KUKA KRL program: EPS_2_25694_WD02A_A_20260120031658.src

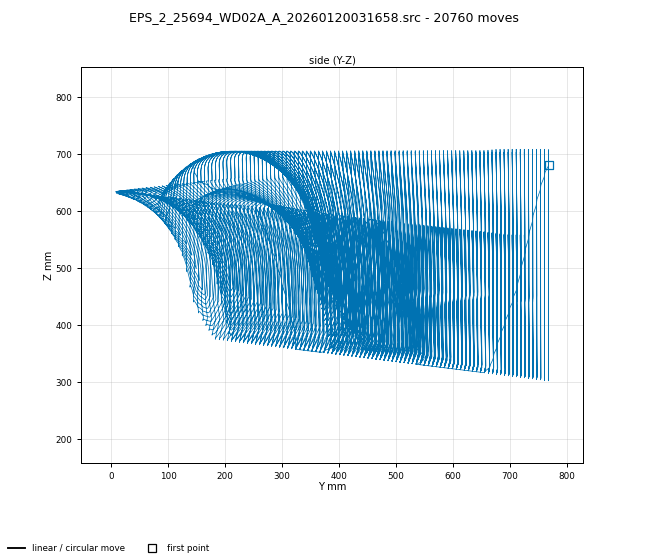
[picture p0: tool path of EPS_2_25694_WD02A_A_20260120031658.src, 20760 of 20762 moves have a stored position in this frame; points joined in program order, loops and branches not executed]
&ACCESS RVP
&REL 4
&COMMENT QRS 19112012
&PARAM EDITMASK = *
DEF PART()
EXT BAS (BAS_COMMAND :IN,REAL :IN )
INT I
BAS (#INITMOV,0 )

;KUKA QRS Post kuka4.cps  Date:22-06-2017 !

File_ID=2999

QRS_PRE_INIT()

;Init var - Until changes are made in qrs_pre_init
Outlet_Square_prg=0
Inlet_1_Square_prg=0
Inlet_2_Square_prg=0
Inlet_3_Square_prg=0
Inlet_4_Square_prg=0
Inlet_5_Square_prg=0

Outlet_1={X 0.000, Y 677.830, Z 583.000, B 0.000, E1 0.000 }
Inlet_1={X 0.000, Y 678.190, Z 578.000, B 0.000, E1 90.000 }
Inlet_2={X 0.000, Y 702.050, Z 243.000, B 0.000, E1 185.000 }
Inlet_3={X 0.000, Y 689.940, Z 413.000, B 0.000, E1 269.000 }
Outlet_1_type=251
Inlet_1_type=251
Inlet_2_type=251
Inlet_3_type=251
;QRS#1=Sidecore dimensions
;QRS#2=250-10" PVC SDR 35
;QRS#3=250-10" PVC SDR 35
;QRS#4=250-10" PVC SDR 35
;QRS#5=250-10" PVC SDR 35
;QRS#6=
;QRS#7=
;QRS#8=
;QRS#9=14M PSX
;QRS#10=14M PSX
;QRS#11=14M PSX
;QRS#12=14M PSX
;QRS#13=
;QRS#14=
;QRS#15=
;QRS#16=1524x152x1067 3,5'
;QRS#17=EPS Height
;QRS#18=708,5
;QRS#19=*
;QRS#20= UPDATED VERSION 22-06-2017
;QRS#21=*
Outlet_Square=0100
Inlet_1_Square=0100
Inlet_2_Square=0100
Inlet_3_Square=0100
Inlet_4_Square=0
Inlet_5_Square=0
Mill_Square=1
Outlet_Square_Prg=205
Inlet_1_Square_prg=205
Inlet_2_Square_prg=205
Inlet_3_Square_prg=205

QRS_INIT()

$ADVANCE=5

; T1
PTP {E1 174.14,E2 174.14}
PTP {X 0,Y 767.497,A -85,B 0,C 180,E1 174.14,E2 174.14,E3 0,E4 0,E5 0,E6 0}
QRS_SPEED_INIT()
LIN {X 0,Y 767.497,Z 681.413,A -85,B 0,C 180,E1 174.14,E2 174.14,E3 0,E4 0,E5 0,E6 0} C_VEL
LIN {X 0,Y 767.498,Z 672.873,A -85,B 0,C 180,E1 173.186,E2 173.186} C_VEL
LIN {X 0,Y 767.497,Z 664.244,A -85,B 0,C 180,E1 172.395,E2 172.395} C_VEL
LIN {X 0,Y 767.496,Z 653.783,A -85,B 0,C 180,E1 171.603,E2 171.603} C_VEL
LIN {X 0,Y 767.499,Z 642.079,A -85,B 0,C 180,E1 170.876,E2 170.876} C_VEL
LIN {X 0,Y 767.47,Z 630.607,A -85,B 0,C 180,E1 170.293,E2 170.293} C_VEL
LIN {X 0,Y 767.488,Z 617.302,A -85,B 0,C 180,E1 169.749,E2 169.749} C_VEL
LIN {X 0,Y 767.494,Z 603.561,A -85,B 0,C 180,E1 169.317,E2 169.317} C_VEL
LIN {X 0,Y 767.478,Z 589.003,A -85,B 0,C 180,E1 168.984,E2 168.984} C_VEL
LIN {X 0,Y 767.456,Z 574.427,A -85,B 0,C 180,E1 168.767,E2 168.767} C_VEL
LIN {X 0,Y 767.491,Z 439.361,A -85,B 0,C 180,E1 167.481,E2 167.481} C_VEL
LIN {X 0,Y 767.485,Z 408.929,A -85,B 0,C 180,E1 164.924,E2 164.924} C_VEL
LIN {X 0,Y 767.474,Z 380.059,A -85,B 0,C 180,E1 162.471,E2 162.471} C_VEL
LIN {X 0,Y 767.471,Z 352.015,A -85,B 0,C 180,E1 160.06,E2 160.06} C_VEL
LIN {X 0,Y 767.448,Z 322.254,A -85,B 0,C 180,E1 157.46,E2 157.46} C_VEL
LIN {X 0,Y 767.468,Z 302.31,A -85,B 0,C 180,E1 155.679,E2 155.679} C_VEL
LIN {X 0,Y 767.445,Z 302.313,A -85,B 0,C 180,E1 153.434,E2 153.434} C_VEL
LIN {X 0,Y 767.444,Z 302.316,A -85,B 0,C 180,E1 151.186,E2 151.186} C_VEL
LIN {X 0,Y 767.451,Z 302.319,A -85,B 0,C 180,E1 149.085,E2 149.085} C_VEL
LIN {X 0,Y 767.479,Z 302.325,A -85,B 0,C 180,E1 146.798,E2 146.798} C_VEL
LIN {X 0,Y 767.488,Z 302.309,A -85,B 0,C 180,E1 144.261,E2 144.261} C_VEL
LIN {X 0,Y 767.459,Z 302.311,A -85,B 0,C 180,E1 141.712,E2 141.712} C_VEL
LIN {X 0,Y 767.472,Z 302.32,A -85,B 0,C 180,E1 139.245,E2 139.245} C_VEL
LIN {X 0,Y 767.481,Z 302.319,A -85,B 0,C 180,E1 136.804,E2 136.804} C_VEL
LIN {X 0,Y 767.479,Z 302.311,A -85,B 0,C 180,E1 134.612,E2 134.612} C_VEL
LIN {X 0,Y 767.493,Z 302.302,A -85,B 0,C 180,E1 132.333,E2 132.333} C_VEL
LIN {X 0,Y 767.47,Z 302.31,A -85,B 0,C 180,E1 129.946,E2 129.946} C_VEL
LIN {X 0,Y 767.489,Z 302.325,A -85,B 0,C 180,E1 127.439,E2 127.439} C_VEL
LIN {X 0,Y 767.472,Z 302.317,A -85,B 0,C 180,E1 125.098,E2 125.098} C_VEL
LIN {X 0,Y 767.487,Z 302.303,A -85,B 0,C 180,E1 122.579,E2 122.579} C_VEL
LIN {X 0,Y 767.485,Z 302.319,A -85,B 0,C 180,E1 119.886,E2 119.886} C_VEL
LIN {X 0,Y 767.49,Z 302.326,A -85,B 0,C 180,E1 117.715,E2 117.715} C_VEL
LIN {X 0,Y 767.461,Z 302.317,A -85,B 0,C 180,E1 115.37,E2 115.37} C_VEL
LIN {X 0,Y 767.457,Z 302.311,A -85,B 0,C 180,E1 113.107,E2 113.107} C_VEL
LIN {X 0,Y 767.471,Z 302.307,A -85,B 0,C 180,E1 110.851,E2 110.851} C_VEL
LIN {X 0,Y 767.488,Z 302.316,A -85,B 0,C 180,E1 108.349,E2 108.349} C_VEL
LIN {X 0,Y 767.466,Z 302.321,A -85,B 0,C 180,E1 105.891,E2 105.891} C_VEL
LIN {X 0,Y 767.447,Z 302.319,A -85,B 0,C 180,E1 103.727,E2 103.727} C_VEL
LIN {X 0,Y 767.436,Z 302.317,A -85,B 0,C 180,E1 101.583,E2 101.583} C_VEL
LIN {X 0,Y 767.437,Z 302.315,A -85,B 0,C 180,E1 99.456,E2 99.456} C_VEL
LIN {X 0,Y 767.443,Z 302.314,A -85,B 0,C 180,E1 97.341,E2 97.341} C_VEL
LIN {X 0,Y 767.498,Z 433.19,A -85,B 0,C 180,E1 96.1,E2 96.1} C_VEL
LIN {X 0,Y 767.498,Z 447.457,A -85,B 0,C 180,E1 95.859,E2 95.859} C_VEL
LIN {X 0,Y 767.489,Z 460.767,A -85,B 0,C 180,E1 95.532,E2 95.532} C_VEL
LIN {X 0,Y 767.487,Z 473.794,A -85,B 0,C 180,E1 95.105,E2 95.105} C_VEL
LIN {X 0,Y 767.483,Z 486.382,A -85,B 0,C 180,E1 94.58,E2 94.58} C_VEL
LIN {X 0,Y 767.496,Z 498.984,A -85,B 0,C 180,E1 93.925,E2 93.925} C_VEL
LIN {X 0,Y 767.499,Z 509.318,A -85,B 0,C 180,E1 93.27,E2 93.27} C_VEL
LIN {X 0,Y 767.497,Z 519.611,A -85,B 0,C 180,E1 92.484,E2 92.484} C_VEL
LIN {X 0,Y 767.498,Z 528.122,A -85,B 0,C 180,E1 91.7,E2 91.7} C_VEL
LIN {X 0,Y 767.497,Z 536.3,A -85,B 0,C 180,E1 90.784,E2 90.784} C_VEL
LIN {X 0,Y 767.497,Z 542.011,A -85,B 0,C 180,E1 90,E2 90} C_VEL
LIN {X 0,Y 767.491,Z 548.132,A -85,B 0,C 180,E1 88.954,E2 88.954} C_VEL
LIN {X 0,Y 767.497,Z 552.64,A -85,B 0,C 180,E1 87.908,E2 87.908} C_VEL
LIN {X 0,Y 767.495,Z 555.711,A -85,B 0,C 180,E1 86.861,E2 86.861} C_VEL
LIN {X 0,Y 767.498,Z 557.427,A -85,B 0,C 180,E1 85.813,E2 85.813} C_VEL
LIN {X 0,Y 767.491,Z 557.838,A -85,B 0,C 180,E1 84.764,E2 84.764} C_VEL
LIN {X 0,Y 767.494,Z 556.939,A -85,B 0,C 180,E1 83.712,E2 83.712} C_VEL
LIN {X 0,Y 767.492,Z 554.711,A -85,B 0,C 180,E1 82.659,E2 82.659} C_VEL
LIN {X 0,Y 767.498,Z 551.074,A -85,B 0,C 180,E1 81.603,E2 81.603} C_VEL
LIN {X 0,Y 767.493,Z 545.927,A -85,B 0,C 180,E1 80.545,E2 80.545} C_VEL
LIN {X 0,Y 767.497,Z 540.906,A -85,B 0,C 180,E1 79.749,E2 79.749} C_VEL
LIN {X 0,Y 767.497,Z 533.708,A -85,B 0,C 180,E1 78.817,E2 78.817} C_VEL
LIN {X 0,Y 767.496,Z 526.139,A -85,B 0,C 180,E1 78.017,E2 78.017} C_VEL
LIN {X 0,Y 767.499,Z 517.02,A -85,B 0,C 180,E1 77.214,E2 77.214} C_VEL
LIN {X 0,Y 767.497,Z 507.896,A -85,B 0,C 180,E1 76.542,E2 76.542} C_VEL
LIN {X 0,Y 767.498,Z 496.967,A -85,B 0,C 180,E1 75.869,E2 75.869} C_VEL
LIN {X 0,Y 767.496,Z 484.947,A -85,B 0,C 180,E1 75.262,E2 75.262} C_VEL
LIN {X 0,Y 767.469,Z 473.355,A -85,B 0,C 180,E1 74.788,E2 74.788} C_VEL
LIN {X 0,Y 767.486,Z 459.725,A -85,B 0,C 180,E1 74.347,E2 74.347} C_VEL
LIN {X 0,Y 767.499,Z 445.316,A -85,B 0,C 180,E1 74.008,E2 74.008} C_VEL
LIN {X 0,Y 767.498,Z 431.17,A -85,B 0,C 180,E1 73.787,E2 73.787} C_VEL
LIN {X 0,Y 767.405,Z 302.321,A -85,B 0,C 180,E1 72.555,E2 72.555} C_VEL
LIN {X 0,Y 767.424,Z 302.32,A -85,B 0,C 180,E1 70.817,E2 70.817} C_VEL
LIN {X 0,Y 767.407,Z 302.321,A -85,B 0,C 180,E1 68.586,E2 68.586} C_VEL
LIN {X 0,Y 767.425,Z 302.32,A -85,B 0,C 180,E1 66.892,E2 66.892} C_VEL
LIN {X 0,Y 767.405,Z 302.321,A -85,B 0,C 180,E1 64.638,E2 64.638} C_VEL
LIN {X 0,Y 767.416,Z 302.32,A -85,B 0,C 180,E1 62.847,E2 62.847} C_VEL
LIN {X 0,Y 767.434,Z 302.319,A -85,B 0,C 180,E1 61.07,E2 61.07} C_VEL
LIN {X 0,Y 767.432,Z 302.319,A -85,B 0,C 180,E1 59.088,E2 59.088} C_VEL
LIN {X 0,Y 767.408,Z 302.321,A -85,B 0,C 180,E1 56.794,E2 56.794} C_VEL
LIN {X 0,Y 767.411,Z 302.32,A -85,B 0,C 180,E1 54.898,E2 54.898} C_VEL
LIN {X 0,Y 767.413,Z 302.32,A -85,B 0,C 180,E1 52.957,E2 52.957} C_VEL
LIN {X 0,Y 767.408,Z 302.321,A -85,B 0,C 180,E1 50.881,E2 50.881} C_VEL
LIN {X 0,Y 767.408,Z 302.321,A -85,B 0,C 180,E1 48.915,E2 48.915} C_VEL
LIN {X 0,Y 767.404,Z 302.321,A -85,B 0,C 180,E1 46.903,E2 46.903} C_VEL
LIN {X 0,Y 767.409,Z 302.322,A -85,B 0,C 180,E1 44.653,E2 44.653} C_VEL
LIN {X 0,Y 767.41,Z 302.32,A -85,B 0,C 180,E1 43.097,E2 43.097} C_VEL
LIN {X 0,Y 767.41,Z 302.32,A -85,B 0,C 180,E1 41.085,E2 41.085} C_VEL
LIN {X 0,Y 767.41,Z 302.32,A -85,B 0,C 180,E1 39.12,E2 39.12} C_VEL
LIN {X 0,Y 767.407,Z 302.321,A -85,B 0,C 180,E1 37.043,E2 37.043} C_VEL
LIN {X 0,Y 767.408,Z 302.32,A -85,B 0,C 180,E1 35.102,E2 35.102} C_VEL
LIN {X 0,Y 767.41,Z 302.32,A -85,B 0,C 180,E1 33.206,E2 33.206} C_VEL
LIN {X 0,Y 767.416,Z 302.32,A -85,B 0,C 180,E1 31.35,E2 31.35} C_VEL
LIN {X 0,Y 767.428,Z 302.319,A -85,B 0,C 180,E1 29.529,E2 29.529} C_VEL
LIN {X 0,Y 767.441,Z 302.319,A -85,B 0,C 180,E1 27.708,E2 27.708} C_VEL
LIN {X 0,Y 767.412,Z 302.32,A -85,B 0,C 180,E1 25.363,E2 25.363} C_VEL
LIN {X 0,Y 767.434,Z 302.318,A -85,B 0,C 180,E1 23.678,E2 23.678} C_VEL
LIN {X 0,Y 767.411,Z 302.32,A -85,B 0,C 180,E1 21.409,E2 21.409} C_VEL
LIN {X 0,Y 767.433,Z 302.318,A -85,B 0,C 180,E1 19.737,E2 19.737} C_VEL
LIN {X 0,Y 767.476,Z 302.317,A -85,B 0,C 180,E1 18.078,E2 18.078} C_VEL
LIN {X 0,Y 767.444,Z 302.318,A -85,B 0,C 180,E1 15.891,E2 15.891} C_VEL
LIN {X 0,Y 767.423,Z 302.319,A -85,B 0,C 180,E1 13.728,E2 13.728} C_VEL
LIN {X 0,Y 767.408,Z 302.321,A -85,B 0,C 180,E1 13.342,E2 13.342} C_VEL
LIN {X 0,Y 767.497,Z 433.16,A -85,B 0,C 180,E1 12.1,E2 12.1} C_VEL
LIN {X 0,Y 767.497,Z 447.876,A -85,B 0,C 180,E1 11.85,E2 11.85} C_VEL
LIN {X 0,Y 767.488,Z 461.291,A -85,B 0,C 180,E1 11.516,E2 11.516} C_VEL
LIN {X 0,Y 767.482,Z 475.246,A -85,B 0,C 180,E1 11.05,E2 11.05} C_VEL
LIN {X 0,Y 767.492,Z 487.712,A -85,B 0,C 180,E1 10.517,E2 10.517} C_VEL
LIN {X 0,Y 767.497,Z 499.092,A -85,B 0,C 180,E1 9.919,E2 9.919} C_VEL
LIN {X 0,Y 767.498,Z 510.478,A -85,B 0,C 180,E1 9.19,E2 9.19} C_VEL
LIN {X 0,Y 767.499,Z 520.651,A -85,B 0,C 180,E1 8.397,E2 8.397} C_VEL
LIN {X 0,Y 767.497,Z 529.057,A -85,B 0,C 180,E1 7.605,E2 7.605} C_VEL
LIN {X 0,Y 767.493,Z 537.081,A -85,B 0,C 180,E1 6.682,E2 6.682} C_VEL
LIN {X 0,Y 767.491,Z 543.547,A -85,B 0,C 180,E1 5.762,E2 5.762} C_VEL
LIN {X 0,Y 767.499,Z 549.276,A -85,B 0,C 180,E1 4.712,E2 4.712} C_VEL
LIN {X 0,Y 767.495,Z 553.459,A -85,B 0,C 180,E1 3.663,E2 3.663} C_VEL
LIN {X 0,Y 767.495,Z 556.221,A -85,B 0,C 180,E1 2.616,E2 2.616} C_VEL
LIN {X 0,Y 767.491,Z 557.643,A -85,B 0,C 180,E1 1.569,E2 1.569} C_VEL
LIN {X 0,Y 767.494,Z 557.768,A -85,B 0,C 180,E1 0.523,E2 0.523} C_VEL
LIN {X 0,Y 767.495,Z 556.591,A -85,B 0,C 180,E1 -0.523,E2 -0.523} C_VEL
LIN {X 0,Y 767.499,Z 554.075,A -85,B 0,C 180,E1 -1.569,E2 -1.569} C_VEL
LIN {X 0,Y 767.493,Z 550.148,A -85,B 0,C 180,E1 -2.615,E2 -2.615} C_VEL
LIN {X 0,Y 767.492,Z 544.699,A -85,B 0,C 180,E1 -3.663,E2 -3.663} C_VEL
LIN {X 0,Y 767.496,Z 539.543,A -85,B 0,C 180,E1 -4.449,E2 -4.449} C_VEL
LIN {X 0,Y 767.496,Z 532.105,A -85,B 0,C 180,E1 -5.367,E2 -5.367} C_VEL
LIN {X 0,Y 767.499,Z 524.084,A -85,B 0,C 180,E1 -6.18,E2 -6.18} C_VEL
LIN {X 0,Y 767.499,Z 515.008,A -85,B 0,C 180,E1 -6.945,E2 -6.945} C_VEL
LIN {X 0,Y 767.498,Z 503.608,A -85,B 0,C 180,E1 -7.736,E2 -7.736} C_VEL
LIN {X 0,Y 767.498,Z 491.988,A -85,B 0,C 180,E1 -8.396,E2 -8.396} C_VEL
LIN {X 0,Y 767.493,Z 479.052,A -85,B 0,C 180,E1 -8.991,E2 -8.991} C_VEL
LIN {X 0,Y 767.495,Z 466.313,A -85,B 0,C 180,E1 -9.455,E2 -9.455} C_VEL
LIN {X 0,Y 767.498,Z 453.375,A -85,B 0,C 180,E1 -9.817,E2 -9.817} C_VEL
LIN {X 0,Y 767.496,Z 439.228,A -85,B 0,C 180,E1 -10.102,E2 -10.102} C_VEL
LIN {X 0,Y 767.498,Z 424.424,A -85,B 0,C 180,E1 -10.284,E2 -10.284} C_VEL
LIN {X 0,Y 767.484,Z 302.305,A -85,B 0,C 180,E1 -11.433,E2 -11.433} C_VEL
LIN {X 0,Y 767.464,Z 302.311,A -85,B 0,C 180,E1 -13.727,E2 -13.727} C_VEL
LIN {X 0,Y 767.467,Z 302.315,A -85,B 0,C 180,E1 -15.89,E2 -15.89} C_VEL
LIN {X 0,Y 767.491,Z 302.323,A -85,B 0,C 180,E1 -18.35,E2 -18.35} C_VEL
LIN {X 0,Y 767.477,Z 302.308,A -85,B 0,C 180,E1 -20.851,E2 -20.851} C_VEL
LIN {X 0,Y 767.486,Z 302.304,A -85,B 0,C 180,E1 -23.106,E2 -23.106} C_VEL
LIN {X 0,Y 767.48,Z 302.31,A -85,B 0,C 180,E1 -25.401,E2 -25.401} C_VEL
LIN {X 0,Y 767.492,Z 302.322,A -85,B 0,C 180,E1 -27.739,E2 -27.739} C_VEL
LIN {X 0,Y 767.464,Z 302.318,A -85,B 0,C 180,E1 -30.13,E2 -30.13} C_VEL
LIN {X 0,Y 767.461,Z 302.31,A -85,B 0,C 180,E1 -32.58,E2 -32.58} C_VEL
LIN {X 0,Y 767.487,Z 302.312,A -85,B 0,C 180,E1 -35.097,E2 -35.097} C_VEL
LIN {X 0,Y 767.465,Z 302.322,A -85,B 0,C 180,E1 -37.697,E2 -37.697} C_VEL
LIN {X 0,Y 767.44,Z 302.318,A -85,B 0,C 180,E1 -39.944,E2 -39.944} C_VEL
LIN {X 0,Y 767.441,Z 302.32,A -85,B 0,C 180,E1 -41.78,E2 -41.78} C_VEL
LIN {X 0,Y 767.429,Z 302.318,A -85,B 0,C 180,E1 -43.921,E2 -43.921} C_VEL
LIN {X 0,Y 767.428,Z 302.317,A -85,B 0,C 180,E1 -46.141,E2 -46.141} C_VEL
LIN {X 0,Y 767.459,Z 302.316,A -85,B 0,C 180,E1 -48.452,E2 -48.452} C_VEL
LIN {X 0,Y 767.48,Z 302.325,A -85,B 0,C 180,E1 -50.969,E2 -50.969} C_VEL
LIN {X 0,Y 767.464,Z 302.325,A -85,B 0,C 180,E1 -52.96,E2 -52.96} C_VEL
LIN {X 0,Y 767.417,Z 302.324,A -85,B 0,C 180,E1 -55.231,E2 -55.231} C_VEL
LIN {X 0,Y 767.395,Z 302.325,A -85,B 0,C 180,E1 -57.416,E2 -57.416} C_VEL
LIN {X 0,Y 767.4,Z 302.325,A -85,B 0,C 180,E1 -59.26,E2 -59.26} C_VEL
LIN {X 0,Y 767.404,Z 302.324,A -85,B 0,C 180,E1 -61.192,E2 -61.192} C_VEL
LIN {X 0,Y 767.435,Z 302.322,A -85,B 0,C 180,E1 -62.848,E2 -62.848} C_VEL
LIN {X 0,Y 767.41,Z 302.321,A -85,B 0,C 180,E1 -65.174,E2 -65.174} C_VEL
LIN {X 0,Y 767.414,Z 302.419,A -85,B 0,C 180,E1 -65.534,E2 -65.534} C_VEL
LIN {X 0,Y 767.485,Z 327.757,A -85,B 0,C 180,E1 -67.744,E2 -67.744} C_VEL
LIN {X 0,Y 767.493,Z 358.817,A -85,B 0,C 180,E1 -70.403,E2 -70.403} C_VEL
LIN {X 0,Y 767.479,Z 388.23,A -85,B 0,C 180,E1 -72.882,E2 -72.882} C_VEL
LIN {X 0,Y 767.425,Z 414.354,A -85,B 0,C 180,E1 -75.058,E2 -75.058} C_VEL
LIN {X 0,Y 767.448,Z 440.449,A -85,B 0,C 180,E1 -77.213,E2 -77.213} C_VEL
LIN {X 0,Y 767.479,Z 444.392,A -85,B 0,C 180,E1 -77.537,E2 -77.537} C_VEL
LIN {X 0,Y 767.465,Z 582.855,A -85,B 0,C 180,E1 -78.85,E2 -78.85} C_VEL
LIN {X 0,Y 767.479,Z 596.903,A -85,B 0,C 180,E1 -79.083,E2 -79.083} C_VEL
LIN {X 0,Y 767.487,Z 610.534,A -85,B 0,C 180,E1 -79.416,E2 -79.416} C_VEL
LIN {X 0,Y 767.478,Z 622.88,A -85,B 0,C 180,E1 -79.815,E2 -79.815} C_VEL
LIN {X 0,Y 767.493,Z 635.798,A -85,B 0,C 180,E1 -80.347,E2 -80.347} C_VEL
LIN {X 0,Y 767.499,Z 647.449,A -85,B 0,C 180,E1 -80.942,E2 -80.942} C_VEL
LIN {X 0,Y 767.496,Z 658.128,A -85,B 0,C 180,E1 -81.603,E2 -81.603} C_VEL
LIN {X 0,Y 767.498,Z 668.693,A -85,B 0,C 180,E1 -82.396,E2 -82.396} C_VEL
LIN {X 0,Y 767.497,Z 677.413,A -85,B 0,C 180,E1 -83.186,E2 -83.186} C_VEL
LIN {X 0,Y 767.497,Z 684.241,A -85,B 0,C 180,E1 -83.926,E2 -83.926} C_VEL
LIN {X 0,Y 767.497,Z 690.701,A -85,B 0,C 180,E1 -84.764,E2 -84.764} C_VEL
LIN {X 0,Y 767.495,Z 697.123,A -85,B 0,C 180,E1 -85.813,E2 -85.813} C_VEL
LIN {X 0,Y 767.495,Z 701.924,A -85,B 0,C 180,E1 -86.861,E2 -86.861} C_VEL
LIN {X 0,Y 767.497,Z 705.261,A -85,B 0,C 180,E1 -87.908,E2 -87.908} C_VEL
LIN {X 0,Y 767.491,Z 707.231,A -85,B 0,C 180,E1 -88.954,E2 -88.954} C_VEL
LIN {X 0,Y 767.494,Z 707.889,A -85,B 0,C 180,E1 -90,E2 -90} C_VEL
LIN {X 0,Y 767.491,Z 707.231,A -85,B 0,C 180,E1 -91.046,E2 -91.046} C_VEL
LIN {X 0,Y 767.497,Z 705.262,A -85,B 0,C 180,E1 -92.092,E2 -92.092} C_VEL
LIN {X 0,Y 767.495,Z 701.925,A -85,B 0,C 180,E1 -93.139,E2 -93.139} C_VEL
LIN {X 0,Y 767.492,Z 697.125,A -85,B 0,C 180,E1 -94.187,E2 -94.187} C_VEL
LIN {X 0,Y 767.497,Z 690.702,A -85,B 0,C 180,E1 -95.236,E2 -95.236} C_VEL
LIN {X 0,Y 767.497,Z 684.242,A -85,B 0,C 180,E1 -96.074,E2 -96.074} C_VEL
LIN {X 0,Y 767.498,Z 676.066,A -85,B 0,C 180,E1 -96.945,E2 -96.945} C_VEL
LIN {X 0,Y 767.498,Z 667.082,A -85,B 0,C 180,E1 -97.736,E2 -97.736} C_VEL
LIN {X 0,Y 767.498,Z 656.192,A -85,B 0,C 180,E1 -98.529,E2 -98.529} C_VEL
LIN {X 0,Y 767.498,Z 645.078,A -85,B 0,C 180,E1 -99.19,E2 -99.19} C_VEL
LIN {X 0,Y 767.497,Z 632.836,A -85,B 0,C 180,E1 -99.785,E2 -99.785} C_VEL
LIN {X 0,Y 767.477,Z 621,A -85,B 0,C 180,E1 -100.251,E2 -100.251} C_VEL
LIN {X 0,Y 767.487,Z 608.116,A -85,B 0,C 180,E1 -100.65,E2 -100.65} C_VEL
LIN {X 0,Y 767.477,Z 595.195,A -85,B 0,C 180,E1 -100.95,E2 -100.95} C_VEL
LIN {X 0,Y 767.464,Z 581.392,A -85,B 0,C 180,E1 -101.166,E2 -101.166} C_VEL
LIN {X 0,Y 767.483,Z 444.379,A -85,B 0,C 180,E1 -102.463,E2 -102.463} C_VEL
LIN {X 0,Y 767.426,Z 417.866,A -85,B 0,C 180,E1 -104.651,E2 -104.651} C_VEL
LIN {X 0,Y 767.447,Z 392.168,A -85,B 0,C 180,E1 -106.789,E2 -106.789} C_VEL
LIN {X 0,Y 767.487,Z 365.358,A -85,B 0,C 180,E1 -109.043,E2 -109.043} C_VEL
LIN {X 0,Y 767.487,Z 335.841,A -85,B 0,C 180,E1 -111.56,E2 -111.56} C_VEL
LIN {X 0,Y 767.445,Z 306.361,A -85,B 0,C 180,E1 -114.119,E2 -114.119} C_VEL
LIN {X 0,Y 767.413,Z 302.322,A -85,B 0,C 180,E1 -114.484,E2 -114.484} C_VEL
LIN {X 0,Y 767.406,Z 302.322,A -85,B 0,C 180,E1 -116.567,E2 -116.567} C_VEL
LIN {X 0,Y 767.41,Z 302.323,A -85,B 0,C 180,E1 -118.335,E2 -118.335} C_VEL
LIN {X 0,Y 767.419,Z 302.324,A -85,B 0,C 180,E1 -120.132,E2 -120.132} C_VEL
LIN {X 0,Y 767.429,Z 302.324,A -85,B 0,C 180,E1 -121.963,E2 -121.963} C_VEL
LIN {X 0,Y 767.436,Z 302.325,A -85,B 0,C 180,E1 -123.843,E2 -123.843} C_VEL
LIN {X 0,Y 767.441,Z 302.325,A -85,B 0,C 180,E1 -125.742,E2 -125.742} C_VEL
LIN {X 0,Y 767.44,Z 302.325,A -85,B 0,C 180,E1 -127.699,E2 -127.699} C_VEL
LIN {X 0,Y 767.41,Z 302.324,A -85,B 0,C 180,E1 -129.941,E2 -129.941} C_VEL
LIN {X 0,Y 767.422,Z 302.323,A -85,B 0,C 180,E1 -131.781,E2 -131.781} C_VEL
LIN {X 0,Y 767.408,Z 302.323,A -85,B 0,C 180,E1 -133.922,E2 -133.922} C_VEL
LIN {X 0,Y 767.404,Z 302.322,A -85,B 0,C 180,E1 -136.077,E2 -136.077} C_VEL
LIN {X 0,Y 767.406,Z 302.322,A -85,B 0,C 180,E1 -138.218,E2 -138.218} C_VEL
LIN {X 0,Y 767.41,Z 302.321,A -85,B 0,C 180,E1 -140.059,E2 -140.059} C_VEL
LIN {X 0,Y 767.423,Z 302.319,A -85,B 0,C 180,E1 -141.715,E2 -141.715} C_VEL
LIN {X 0,Y 767.431,Z 302.318,A -85,B 0,C 180,E1 -143.611,E2 -143.611} C_VEL
LIN {X 0,Y 767.436,Z 302.317,A -85,B 0,C 180,E1 -145.537,E2 -145.537} C_VEL
LIN {X 0,Y 767.445,Z 302.315,A -85,B 0,C 180,E1 -147.419,E2 -147.419} C_VEL
LIN {X 0,Y 767.461,Z 302.313,A -85,B 0,C 180,E1 -149.263,E2 -149.263} C_VEL
LIN {X 0,Y 767.428,Z 302.317,A -85,B 0,C 180,E1 -151.666,E2 -151.666} C_VEL
LIN {X 0,Y 767.439,Z 302.314,A -85,B 0,C 180,E1 -153.438,E2 -153.438} C_VEL
LIN {X 0,Y 767.462,Z 302.311,A -85,B 0,C 180,E1 -155.176,E2 -155.176} C_VEL
LIN {X 0,Y 767.433,Z 302.347,A -85,B 0,C 180,E1 -155.783,E2 -155.783} C_VEL
LIN {X 0,Y 767.491,Z 327.656,A -85,B 0,C 180,E1 -158.026,E2 -158.026} C_VEL
LIN {X 0,Y 767.472,Z 356.548,A -85,B 0,C 180,E1 -160.542,E2 -160.542} C_VEL
LIN {X 0,Y 767.484,Z 388.736,A -85,B 0,C 180,E1 -163.301,E2 -163.301} C_VEL
LIN {X 0,Y 767.476,Z 417.477,A -85,B 0,C 180,E1 -165.734,E2 -165.734} C_VEL
LIN {X 0,Y 767.494,Z 439.485,A -85,B 0,C 180,E1 -167.581,E2 -167.581} C_VEL
LIN {X 0,Y 767.493,Z 578.248,A -85,B 0,C 180,E1 -168.901,E2 -168.901} C_VEL
LIN {X 0,Y 767.497,Z 592.889,A -85,B 0,C 180,E1 -169.151,E2 -169.151} C_VEL
LIN {X 0,Y 767.478,Z 606.264,A -85,B 0,C 180,E1 -169.483,E2 -169.483} C_VEL
LIN {X 0,Y 767.448,Z 620.19,A -85,B 0,C 180,E1 -169.947,E2 -169.947} C_VEL
LIN {X 0,Y 767.477,Z 632.725,A -85,B 0,C 180,E1 -170.483,E2 -170.483} C_VEL
LIN {X 0,Y 767.499,Z 643.975,A -85,B 0,C 180,E1 -171.075,E2 -171.075} C_VEL
LIN {X 0,Y 767.496,Z 654.401,A -85,B 0,C 180,E1 -171.736,E2 -171.736} C_VEL
LIN {X 0,Y 767.498,Z 664.759,A -85,B 0,C 180,E1 -172.528,E2 -172.528} C_VEL
LIN {X 0,Y 767.497,Z 673.302,A -85,B 0,C 180,E1 -173.318,E2 -173.318} C_VEL
LIN {X 0,Y 767.496,Z 681.478,A -85,B 0,C 180,E1 -174.238,E2 -174.238} C_VEL
LIN {X 0,Y 767.499,Z 687.19,A -85,B 0,C 180,E1 -175.026,E2 -175.026} C_VEL
LIN {X 0,Y 767.496,Z 691.883,A -85,B 0,C 180,E1 -175.813,E2 -175.813} C_VEL
LIN {X 0,Y 767.497,Z 696.744,A -85,B 0,C 180,E1 -176.861,E2 -176.861} C_VEL
LIN {X 0,Y 767.497,Z 700.14,A -85,B 0,C 180,E1 -177.908,E2 -177.908} C_VEL
LIN {X 0,Y 767.497,Z 702.163,A -85,B 0,C 180,E1 -178.954,E2 -178.954} C_VEL
LIN {X 0,Y 767.492,Z 702.882,A -85,B 0,C 180,E1 -180,E2 -180} C_VEL
LIN {X 0,Y 767.497,Z 702.292,A -85,B 0,C 180,E1 -181.046,E2 -181.046} C_VEL
LIN {X 0,Y 767.495,Z 700.384,A -85,B 0,C 180,E1 -182.092,E2 -182.092} C_VEL
LIN {X 0,Y 767.495,Z 697.104,A -85,B 0,C 180,E1 -183.139,E2 -183.139} C_VEL
LIN {X 0,Y 767.497,Z 692.364,A -85,B 0,C 180,E1 -184.187,E2 -184.187} C_VEL
LIN {X 0,Y 767.496,Z 686.008,A -85,B 0,C 180,E1 -185.236,E2 -185.236} C_VEL
LIN {X 0,Y 767.497,Z 681.413,A -85,B 0,C 180,E1 -185.86,E2 -185.86} C_VEL
LIN {X 0,Y 766.815,Z 678.477,A -85,B 0,C 180,E1 -186.232,E2 -186.232} C_VEL
LIN {X 0,Y 763.938,Z 673.407,A -85,B 0,C 180,E1 -186.83,E2 -186.83} C_VEL
LIN {X 0,Y 761.084,Z 667.642,A -85,B 0,C 180,E1 -187.407,E2 -187.407} C_VEL
LIN {X 0,Y 760.463,Z 663.74,A -85,B 0,C 180,E1 -187.744,E2 -187.744} C_VEL
LIN {X 0,Y 760.461,Z 654.058,A -85,B 0,C 180,E1 -188.475,E2 -188.475} C_VEL
LIN {X 0,Y 760.495,Z 643.46,A -85,B 0,C 180,E1 -189.142,E2 -189.142} C_VEL
LIN {X 0,Y 760.469,Z 631.705,A -85,B 0,C 180,E1 -189.753,E2 -189.753} C_VEL
LIN {X 0,Y 760.49,Z 619.206,A -85,B 0,C 180,E1 -190.28,E2 -190.28} C_VEL
LIN {X 0,Y 760.521,Z 606.056,A -85,B 0,C 180,E1 -190.715,E2 -190.715} C_VEL
LIN {X 0,Y 760.525,Z 591.76,A -85,B 0,C 180,E1 -191.068,E2 -191.068} C_VEL
LIN {X 0,Y 760.515,Z 577.555,A -85,B 0,C 180,E1 -191.304,E2 -191.304} C_VEL
LIN {X 0,Y 760.498,Z 439.696,A -85,B 0,C 180,E1 -192.618,E2 -192.618} C_VEL
LIN {X 0,Y 760.525,Z 410.578,A -85,B 0,C 180,E1 -195.081,E2 -195.081} C_VEL
LIN {X 0,Y 760.544,Z 381.671,A -85,B 0,C 180,E1 -197.555,E2 -197.555} C_VEL
LIN {X 0,Y 760.567,Z 352.872,A -85,B 0,C 180,E1 -200.054,E2 -200.054} C_VEL
LIN {X 0,Y 760.604,Z 323.854,A -85,B 0,C 180,E1 -202.612,E2 -202.612} C_VEL
LIN {X 0,Y 760.673,Z 305.299,A -85,B 0,C 180,E1 -204.27,E2 -204.27} C_VEL
LIN {X 0,Y 760.448,Z 303.313,A -85,B 0,C 180,E1 -204.468,E2 -204.468} C_VEL
LIN {X 0,Y 760.417,Z 303.316,A -85,B 0,C 180,E1 -206.831,E2 -206.831} C_VEL
LIN {X 0,Y 760.422,Z 303.317,A -85,B 0,C 180,E1 -208.947,E2 -208.947} C_VEL
LIN {X 0,Y 760.442,Z 303.318,A -85,B 0,C 180,E1 -211.06,E2 -211.06} C_VEL
LIN {X 0,Y 760.47,Z 303.315,A -85,B 0,C 180,E1 -213.549,E2 -213.549} C_VEL
LIN {X 0,Y 760.443,Z 303.311,A -85,B 0,C 180,E1 -216.122,E2 -216.122} C_VEL
LIN {X 0,Y 760.427,Z 303.315,A -85,B 0,C 180,E1 -218.468,E2 -218.468} C_VEL
LIN {X 0,Y 760.446,Z 303.32,A -85,B 0,C 180,E1 -220.843,E2 -220.843} C_VEL
LIN {X 0,Y 760.462,Z 303.314,A -85,B 0,C 180,E1 -223.31,E2 -223.31} C_VEL
LIN {X 0,Y 760.438,Z 303.313,A -85,B 0,C 180,E1 -225.57,E2 -225.57} C_VEL
LIN {X 0,Y 760.457,Z 303.31,A -85,B 0,C 180,E1 -227.748,E2 -227.748} C_VEL
LIN {X 0,Y 760.474,Z 303.308,A -85,B 0,C 180,E1 -229.861,E2 -229.861} C_VEL
LIN {X 0,Y 760.466,Z 303.316,A -85,B 0,C 180,E1 -232.385,E2 -232.385} C_VEL
LIN {X 0,Y 760.44,Z 303.325,A -85,B 0,C 180,E1 -234.529,E2 -234.529} C_VEL
LIN {X 0,Y 760.451,Z 303.314,A -85,B 0,C 180,E1 -236.95,E2 -236.95} C_VEL
LIN {X 0,Y 760.436,Z 303.315,A -85,B 0,C 180,E1 -238.948,E2 -238.948} C_VEL
LIN {X 0,Y 760.443,Z 303.311,A -85,B 0,C 180,E1 -241.382,E2 -241.382} C_VEL
LIN {X 0,Y 760.464,Z 303.313,A -85,B 0,C 180,E1 -243.761,E2 -243.761} C_VEL
LIN {X 0,Y 760.448,Z 303.323,A -85,B 0,C 180,E1 -246.091,E2 -246.091} C_VEL
LIN {X 0,Y 760.432,Z 303.317,A -85,B 0,C 180,E1 -248.486,E2 -248.486} C_VEL
LIN {X 0,Y 760.434,Z 303.314,A -85,B 0,C 180,E1 -250.634,E2 -250.634} C_VEL
LIN {X 0,Y 760.441,Z 303.312,A -85,B 0,C 180,E1 -252.857,E2 -252.857} C_VEL
LIN {X 0,Y 760.463,Z 303.318,A -85,B 0,C 180,E1 -255.6,E2 -255.6} C_VEL
LIN {X 0,Y 760.473,Z 303.32,A -85,B 0,C 180,E1 -257.77,E2 -257.77} C_VEL
LIN {X 0,Y 760.432,Z 303.314,A -85,B 0,C 180,E1 -260.264,E2 -260.264} C_VEL
LIN {X 0,Y 760.419,Z 303.315,A -85,B 0,C 180,E1 -262.541,E2 -262.541} C_VEL
LIN {X 0,Y 760.551,Z 337.066,A -85,B 0,C 180,E1 -262.875,E2 -262.875} C_VEL
LIN {X 0,Y 760.548,Z 433.853,A -85,B 0,C 180,E1 -263.804,E2 -263.804} C_VEL
LIN {X 0,Y 760.529,Z 448.118,A -85,B 0,C 180,E1 -264.051,E2 -264.051} C_VEL
LIN {X 0,Y 760.523,Z 462.041,A -85,B 0,C 180,E1 -264.404,E2 -264.404} C_VEL
LIN {X 0,Y 760.508,Z 475.187,A -85,B 0,C 180,E1 -264.848,E2 -264.848} C_VEL
LIN {X 0,Y 760.473,Z 487.569,A -85,B 0,C 180,E1 -265.377,E2 -265.377} C_VEL
LIN {X 0,Y 760.496,Z 498.889,A -85,B 0,C 180,E1 -265.973,E2 -265.973} C_VEL
LIN {X 0,Y 760.487,Z 510.277,A -85,B 0,C 180,E1 -266.7,E2 -266.7} C_VEL
LIN {X 0,Y 760.48,Z 520.508,A -85,B 0,C 180,E1 -267.493,E2 -267.493} C_VEL
LIN {X 0,Y 760.452,Z 528.978,A -85,B 0,C 180,E1 -268.285,E2 -268.285} C_VEL
LIN {X 0,Y 760.452,Z 537.101,A -85,B 0,C 180,E1 -269.208,E2 -269.208} C_VEL
LIN {X 0,Y 760.441,Z 542.811,A -85,B 0,C 180,E1 -270,E2 -270} C_VEL
LIN {X 0,Y 760.446,Z 548.891,A -85,B 0,C 180,E1 -271.056,E2 -271.056} C_VEL
LIN {X 0,Y 760.425,Z 553.362,A -85,B 0,C 180,E1 -272.112,E2 -272.112} C_VEL
LIN {X 0,Y 760.421,Z 556.4,A -85,B 0,C 180,E1 -273.168,E2 -273.168} C_VEL
LIN {X 0,Y 760.437,Z 558.077,A -85,B 0,C 180,E1 -274.226,E2 -274.226} C_VEL
LIN {X 0,Y 760.429,Z 558.436,A -85,B 0,C 180,E1 -275.285,E2 -275.285} C_VEL
LIN {X 0,Y 760.434,Z 557.475,A -85,B 0,C 180,E1 -276.346,E2 -276.346} C_VEL
LIN {X 0,Y 760.428,Z 555.168,A -85,B 0,C 180,E1 -277.409,E2 -277.409} C_VEL
LIN {X 0,Y 760.428,Z 551.44,A -85,B 0,C 180,E1 -278.475,E2 -278.475} C_VEL
LIN {X 0,Y 760.441,Z 546.171,A -85,B 0,C 180,E1 -279.544,E2 -279.544} C_VEL
LIN {X 0,Y 760.455,Z 541.055,A -85,B 0,C 180,E1 -280.347,E2 -280.347} C_VEL
LIN {X 0,Y 760.444,Z 533.725,A -85,B 0,C 180,E1 -281.288,E2 -281.288} C_VEL
LIN {X 0,Y 760.446,Z 524.617,A -85,B 0,C 180,E1 -282.231,E2 -282.231} C_VEL
LIN {X 0,Y 760.46,Z 515.011,A -85,B 0,C 180,E1 -283.042,E2 -283.042} C_VEL
LIN {X 0,Y 760.496,Z 503.258,A -85,B 0,C 180,E1 -283.855,E2 -283.855} C_VEL
LIN {X 0,Y 760.498,Z 491.853,A -85,B 0,C 180,E1 -284.502,E2 -284.502} C_VEL
LIN {X 0,Y 760.473,Z 479.268,A -85,B 0,C 180,E1 -285.082,E2 -285.082} C_VEL
LIN {X 0,Y 760.495,Z 466.18,A -85,B 0,C 180,E1 -285.56,E2 -285.56} C_VEL
LIN {X 0,Y 760.532,Z 451.941,A -85,B 0,C 180,E1 -285.954,E2 -285.954} C_VEL
LIN {X 0,Y 760.56,Z 437.768,A -85,B 0,C 180,E1 -286.228,E2 -286.228} C_VEL
LIN {X 0,Y 760.542,Z 419.746,A -85,B 0,C 180,E1 -286.434,E2 -286.434} C_VEL
LIN {X 0,Y 760.373,Z 303.32,A -85,B 0,C 180,E1 -287.542,E2 -287.542} C_VEL
LIN {X 0,Y 760.397,Z 303.317,A -85,B 0,C 180,E1 -289.367,E2 -289.367} C_VEL
LIN {X 0,Y 760.392,Z 303.318,A -85,B 0,C 180,E1 -291.621,E2 -291.621} C_VEL
LIN {X 0,Y 760.38,Z 303.319,A -85,B 0,C 180,E1 -293.335,E2 -293.335} C_VEL
LIN {X 0,Y 760.385,Z 303.319,A -85,B 0,C 180,E1 -295.655,E2 -295.655} C_VEL
LIN {X 0,Y 760.424,Z 303.319,A -85,B 0,C 180,E1 -298.02,E2 -298.02} C_VEL
LIN {X 0,Y 760.42,Z 303.325,A -85,B 0,C 180,E1 -300.439,E2 -300.439} C_VEL
LIN {X 0,Y 760.406,Z 303.317,A -85,B 0,C 180,E1 -302.921,E2 -302.921} C_VEL
LIN {X 0,Y 760.399,Z 303.318,A -85,B 0,C 180,E1 -304.932,E2 -304.932} C_VEL
LIN {X 0,Y 760.432,Z 303.315,A -85,B 0,C 180,E1 -306.779,E2 -306.779} C_VEL
LIN {X 0,Y 760.423,Z 303.316,A -85,B 0,C 180,E1 -308.783,E2 -308.783} C_VEL
LIN {X 0,Y 760.41,Z 303.316,A -85,B 0,C 180,E1 -310.945,E2 -310.945} C_VEL
LIN {X 0,Y 760.395,Z 303.317,A -85,B 0,C 180,E1 -312.974,E2 -312.974} C_VEL
LIN {X 0,Y 760.376,Z 303.319,A -85,B 0,C 180,E1 -315.179,E2 -315.179} C_VEL
LIN {X 0,Y 760.394,Z 303.317,A -85,B 0,C 180,E1 -317.026,E2 -317.026} C_VEL
LIN {X 0,Y 760.378,Z 303.319,A -85,B 0,C 180,E1 -319.153,E2 -319.153} C_VEL
LIN {X 0,Y 760.38,Z 303.319,A -85,B 0,C 180,E1 -321.215,E2 -321.215} C_VEL
LIN {X 0,Y 760.389,Z 303.319,A -85,B 0,C 180,E1 -323.266,E2 -323.266} C_VEL
LIN {X 0,Y 760.389,Z 303.318,A -85,B 0,C 180,E1 -325.171,E2 -325.171} C_VEL
LIN {X 0,Y 760.389,Z 303.318,A -85,B 0,C 180,E1 -327.078,E2 -327.078} C_VEL
LIN {X 0,Y 760.398,Z 303.316,A -85,B 0,C 180,E1 -328.946,E2 -328.946} C_VEL
LIN {X 0,Y 760.393,Z 303.318,A -85,B 0,C 180,E1 -331.058,E2 -331.058} C_VEL
LIN {X 0,Y 760.411,Z 303.319,A -85,B 0,C 180,E1 -333.318,E2 -333.318} C_VEL
LIN {X 0,Y 760.43,Z 303.318,A -85,B 0,C 180,E1 -336.09,E2 -336.09} C_VEL
LIN {X 0,Y 760.407,Z 303.316,A -85,B 0,C 180,E1 -338.491,E2 -338.491} C_VEL
LIN {X 0,Y 760.397,Z 303.317,A -85,B 0,C 180,E1 -340.633,E2 -340.633} C_VEL
LIN {X 0,Y 760.412,Z 303.316,A -85,B 0,C 180,E1 -342.303,E2 -342.303} C_VEL
LIN {X 0,Y 760.405,Z 303.316,A -85,B 0,C 180,E1 -344.506,E2 -344.506} C_VEL
LIN {X 0,Y 760.389,Z 303.318,A -85,B 0,C 180,E1 -346.55,E2 -346.55} C_VEL
LIN {X 0,Y 760.547,Z 433.849,A -85,B 0,C 180,E1 -347.804,E2 -347.804} C_VEL
LIN {X 0,Y 760.535,Z 448.344,A -85,B 0,C 180,E1 -348.057,E2 -348.057} C_VEL
LIN {X 0,Y 760.526,Z 462.233,A -85,B 0,C 180,E1 -348.411,E2 -348.411} C_VEL
LIN {X 0,Y 760.505,Z 475.169,A -85,B 0,C 180,E1 -348.848,E2 -348.848} C_VEL
LIN {X 0,Y 760.482,Z 487.719,A -85,B 0,C 180,E1 -349.385,E2 -349.385} C_VEL
LIN {X 0,Y 760.483,Z 500.001,A -85,B 0,C 180,E1 -350.037,E2 -350.037} C_VEL
LIN {X 0,Y 760.471,Z 510.635,A -85,B 0,C 180,E1 -350.724,E2 -350.724} C_VEL
LIN {X 0,Y 760.453,Z 520.887,A -85,B 0,C 180,E1 -351.525,E2 -351.525} C_VEL
LIN {X 0,Y 760.451,Z 529.36,A -85,B 0,C 180,E1 -352.325,E2 -352.325} C_VEL
LIN {X 0,Y 760.44,Z 537.458,A -85,B 0,C 180,E1 -353.255,E2 -353.255} C_VEL
LIN {X 0,Y 760.437,Z 543.985,A -85,B 0,C 180,E1 -354.185,E2 -354.185} C_VEL
LIN {X 0,Y 760.43,Z 549.775,A -85,B 0,C 180,E1 -355.245,E2 -355.245} C_VEL
LIN {X 0,Y 760.442,Z 554.004,A -85,B 0,C 180,E1 -356.303,E2 -356.303} C_VEL
LIN {X 0,Y 760.423,Z 556.8,A -85,B 0,C 180,E1 -357.36,E2 -357.36} C_VEL
LIN {X 0,Y 760.436,Z 558.245,A -85,B 0,C 180,E1 -358.416,E2 -358.416} C_VEL
LIN {X 0,Y 760.44,Z 558.381,A -85,B 0,C 180,E1 -359.472,E2 -359.472} C_VEL
LIN {X 0,Y 760.441,Z 557.203,A -85,B 0,C 180,E1 -360.528,E2 -360.528} C_VEL
LIN {X 0,Y 760.442,Z 554.681,A -85,B 0,C 180,E1 -361.583,E2 -361.583} C_VEL
LIN {X 0,Y 760.424,Z 550.733,A -85,B 0,C 180,E1 -362.64,E2 -362.64} C_VEL
LIN {X 0,Y 760.441,Z 545.253,A -85,B 0,C 180,E1 -363.697,E2 -363.697} C_VEL
LIN {X 0,Y 760.449,Z 539.066,A -85,B 0,C 180,E1 -364.623,E2 -364.623} C_VEL
LIN {X 0,Y 760.449,Z 531.362,A -85,B 0,C 180,E1 -365.55,E2 -365.55} C_VEL
LIN {X 0,Y 760.468,Z 523.331,A -85,B 0,C 180,E1 -366.346,E2 -366.346} C_VEL
LIN {X 0,Y 760.478,Z 513.667,A -85,B 0,C 180,E1 -367.143,E2 -367.143} C_VEL
LIN {X 0,Y 760.486,Z 502.952,A -85,B 0,C 180,E1 -367.875,E2 -367.875} C_VEL
LIN {X 0,Y 760.49,Z 491.103,A -85,B 0,C 180,E1 -368.541,E2 -368.541} C_VEL
LIN {X 0,Y 760.49,Z 479.44,A -85,B 0,C 180,E1 -369.075,E2 -369.075} C_VEL
LIN {X 0,Y 760.518,Z 465.594,A -85,B 0,C 180,E1 -369.579,E2 -369.579} C_VEL
LIN {X 0,Y 760.53,Z 451.556,A -85,B 0,C 180,E1 -369.962,E2 -369.962} C_VEL
LIN {X 0,Y 760.555,Z 437.726,A -85,B 0,C 180,E1 -370.228,E2 -370.228} C_VEL
LIN {X 0,Y 760.545,Z 420.241,A -85,B 0,C 180,E1 -370.43,E2 -370.43} C_VEL
LIN {X 0,Y 760.461,Z 303.31,A -85,B 0,C 180,E1 -371.54,E2 -371.54} C_VEL
LIN {X 0,Y 760.434,Z 303.315,A -85,B 0,C 180,E1 -373.856,E2 -373.856} C_VEL
LIN {X 0,Y 760.438,Z 303.319,A -85,B 0,C 180,E1 -376.041,E2 -376.041} C_VEL
LIN {X 0,Y 760.457,Z 303.319,A -85,B 0,C 180,E1 -378.428,E2 -378.428} C_VEL
LIN {X 0,Y 760.463,Z 303.315,A -85,B 0,C 180,E1 -380.488,E2 -380.488} C_VEL
LIN {X 0,Y 760.448,Z 303.311,A -85,B 0,C 180,E1 -382.913,E2 -382.913} C_VEL
LIN {X 0,Y 760.441,Z 303.312,A -85,B 0,C 180,E1 -385.069,E2 -385.069} C_VEL
LIN {X 0,Y 760.47,Z 303.312,A -85,B 0,C 180,E1 -387.422,E2 -387.422} C_VEL
LIN {X 0,Y 760.449,Z 303.318,A -85,B 0,C 180,E1 -390.022,E2 -390.022} C_VEL
LIN {X 0,Y 760.427,Z 303.315,A -85,B 0,C 180,E1 -392.293,E2 -392.293} C_VEL
LIN {X 0,Y 760.437,Z 303.314,A -85,B 0,C 180,E1 -394.186,E2 -394.186} C_VEL
LIN {X 0,Y 760.446,Z 303.312,A -85,B 0,C 180,E1 -396.778,E2 -396.778} C_VEL
LIN {X 0,Y 760.457,Z 303.32,A -85,B 0,C 180,E1 -399.461,E2 -399.461} C_VEL
LIN {X 0,Y 760.415,Z 303.318,A -85,B 0,C 180,E1 -401.744,E2 -401.744} C_VEL
LIN {X 0,Y 760.424,Z 303.317,A -85,B 0,C 180,E1 -403.697,E2 -403.697} C_VEL
LIN {X 0,Y 760.394,Z 303.318,A -85,B 0,C 180,E1 -405.931,E2 -405.931} C_VEL
LIN {X 0,Y 760.394,Z 303.318,A -85,B 0,C 180,E1 -407.743,E2 -407.743} C_VEL
LIN {X 0,Y 760.392,Z 303.318,A -85,B 0,C 180,E1 -409.868,E2 -409.868} C_VEL
LIN {X 0,Y 760.404,Z 303.316,A -85,B 0,C 180,E1 -411.89,E2 -411.89} C_VEL
LIN {X 0,Y 760.417,Z 303.317,A -85,B 0,C 180,E1 -414.154,E2 -414.154} C_VEL
LIN {X 0,Y 760.414,Z 303.324,A -85,B 0,C 180,E1 -416.449,E2 -416.449} C_VEL
LIN {X 0,Y 760.412,Z 303.32,A -85,B 0,C 180,E1 -418.946,E2 -418.946} C_VEL
LIN {X 0,Y 760.369,Z 303.321,A -85,B 0,C 180,E1 -421.378,E2 -421.378} C_VEL
LIN {X 0,Y 760.386,Z 303.319,A -85,B 0,C 180,E1 -423.321,E2 -423.321} C_VEL
LIN {X 0,Y 760.398,Z 303.44,A -85,B 0,C 180,E1 -425.384,E2 -425.384} C_VEL
LIN {X 0,Y 760.671,Z 311.41,A -85,B 0,C 180,E1 -426.098,E2 -426.098} C_VEL
LIN {X 0,Y 760.6,Z 339.494,A -85,B 0,C 180,E1 -428.552,E2 -428.552} C_VEL
LIN {X 0,Y 760.569,Z 366.991,A -85,B 0,C 180,E1 -430.917,E2 -430.917} C_VEL
LIN {X 0,Y 760.495,Z 393.474,A -85,B 0,C 180,E1 -433.162,E2 -433.162} C_VEL
LIN {X 0,Y 760.446,Z 418.668,A -85,B 0,C 180,E1 -435.274,E2 -435.274} C_VEL
LIN {X 0,Y 760.469,Z 444.499,A -85,B 0,C 180,E1 -437.42,E2 -437.42} C_VEL
LIN {X 0,Y 760.502,Z 583.003,A -85,B 0,C 180,E1 -438.747,E2 -438.747} C_VEL
LIN {X 0,Y 760.51,Z 597.027,A -85,B 0,C 180,E1 -438.982,E2 -438.982} C_VEL
LIN {X 0,Y 760.503,Z 610.671,A -85,B 0,C 180,E1 -439.318,E2 -439.318} C_VEL
LIN {X 0,Y 760.483,Z 623.036,A -85,B 0,C 180,E1 -439.72,E2 -439.72} C_VEL
LIN {X 0,Y 760.505,Z 635.415,A -85,B 0,C 180,E1 -440.23,E2 -440.23} C_VEL
LIN {X 0,Y 760.495,Z 647.683,A -85,B 0,C 180,E1 -440.858,E2 -440.858} C_VEL
LIN {X 0,Y 760.462,Z 658.406,A -85,B 0,C 180,E1 -441.525,E2 -441.525} C_VEL
LIN {X 0,Y 760.453,Z 669.022,A -85,B 0,C 180,E1 -442.325,E2 -442.325} C_VEL
LIN {X 0,Y 760.465,Z 677.792,A -85,B 0,C 180,E1 -443.123,E2 -443.123} C_VEL
LIN {X 0,Y 760.446,Z 685.313,A -85,B 0,C 180,E1 -443.946,E2 -443.946} C_VEL
LIN {X 0,Y 760.435,Z 691.172,A -85,B 0,C 180,E1 -444.715,E2 -444.715} C_VEL
LIN {X 0,Y 760.436,Z 697.643,A -85,B 0,C 180,E1 -445.774,E2 -445.774} C_VEL
LIN {X 0,Y 760.425,Z 702.483,A -85,B 0,C 180,E1 -446.832,E2 -446.832} C_VEL
LIN {X 0,Y 760.426,Z 705.85,A -85,B 0,C 180,E1 -447.888,E2 -447.888} C_VEL
LIN {X 0,Y 760.445,Z 707.835,A -85,B 0,C 180,E1 -448.944,E2 -448.944} C_VEL
LIN {X 0,Y 760.438,Z 708.5,A -85,B 0,C 180,E1 -450,E2 -450} C_VEL
LIN {X 0,Y 760.445,Z 707.835,A -85,B 0,C 180,E1 -451.055,E2 -451.055} C_VEL
LIN {X 0,Y 760.426,Z 705.85,A -85,B 0,C 180,E1 -452.111,E2 -452.111} C_VEL
LIN {X 0,Y 760.425,Z 702.484,A -85,B 0,C 180,E1 -453.168,E2 -453.168} C_VEL
LIN {X 0,Y 760.434,Z 697.644,A -85,B 0,C 180,E1 -454.226,E2 -454.226} C_VEL
LIN {X 0,Y 760.435,Z 691.173,A -85,B 0,C 180,E1 -455.285,E2 -455.285} C_VEL
LIN {X 0,Y 760.453,Z 684.086,A -85,B 0,C 180,E1 -456.2,E2 -456.2} C_VEL
LIN {X 0,Y 760.447,Z 676.439,A -85,B 0,C 180,E1 -457.01,E2 -457.01} C_VEL
LIN {X 0,Y 760.474,Z 667.404,A -85,B 0,C 180,E1 -457.808,E2 -457.808} C_VEL
LIN {X 0,Y 760.471,Z 656.459,A -85,B 0,C 180,E1 -458.608,E2 -458.608} C_VEL
LIN {X 0,Y 760.491,Z 645.302,A -85,B 0,C 180,E1 -459.275,E2 -459.275} C_VEL
LIN {X 0,Y 760.503,Z 633.695,A -85,B 0,C 180,E1 -459.847,E2 -459.847} C_VEL
LIN {X 0,Y 760.512,Z 621.156,A -85,B 0,C 180,E1 -460.346,E2 -460.346} C_VEL
LIN {X 0,Y 760.526,Z 608.255,A -85,B 0,C 180,E1 -460.749,E2 -460.749} C_VEL
LIN {X 0,Y 760.521,Z 594.418,A -85,B 0,C 180,E1 -461.068,E2 -461.068} C_VEL
LIN {X 0,Y 760.502,Z 580.051,A -85,B 0,C 180,E1 -461.287,E2 -461.287} C_VEL
LIN {X 0,Y 760.471,Z 444.479,A -85,B 0,C 180,E1 -462.582,E2 -462.582} C_VEL
LIN {X 0,Y 760.447,Z 418.665,A -85,B 0,C 180,E1 -464.726,E2 -464.726} C_VEL
LIN {X 0,Y 760.495,Z 393.476,A -85,B 0,C 180,E1 -466.838,E2 -466.838} C_VEL
LIN {X 0,Y 760.569,Z 365.358,A -85,B 0,C 180,E1 -469.223,E2 -469.223} C_VEL
LIN {X 0,Y 760.641,Z 335.933,A -85,B 0,C 180,E1 -471.755,E2 -471.755} C_VEL
LIN {X 0,Y 760.642,Z 307.303,A -85,B 0,C 180,E1 -474.265,E2 -474.265} C_VEL
LIN {X 0,Y 760.392,Z 303.32,A -85,B 0,C 180,E1 -474.634,E2 -474.634} C_VEL
LIN {X 0,Y 760.395,Z 303.318,A -85,B 0,C 180,E1 -476.831,E2 -476.831} C_VEL
LIN {X 0,Y 760.393,Z 303.319,A -85,B 0,C 180,E1 -478.943,E2 -478.943} C_VEL
LIN {X 0,Y 760.415,Z 303.318,A -85,B 0,C 180,E1 -481.057,E2 -481.057} C_VEL
LIN {X 0,Y 760.413,Z 303.327,A -85,B 0,C 180,E1 -483.551,E2 -483.551} C_VEL
LIN {X 0,Y 760.393,Z 303.318,A -85,B 0,C 180,E1 -486.125,E2 -486.125} C_VEL
LIN {X 0,Y 760.369,Z 303.321,A -85,B 0,C 180,E1 -488.112,E2 -488.112} C_VEL
LIN {X 0,Y 760.385,Z 303.319,A -85,B 0,C 180,E1 -490.152,E2 -490.152} C_VEL
LIN {X 0,Y 760.372,Z 303.32,A -85,B 0,C 180,E1 -492.258,E2 -492.258} C_VEL
LIN {X 0,Y 760.375,Z 303.32,A -85,B 0,C 180,E1 -494.067,E2 -494.067} C_VEL
LIN {X 0,Y 760.399,Z 303.317,A -85,B 0,C 180,E1 -496.301,E2 -496.301} C_VEL
LIN {X 0,Y 760.41,Z 303.318,A -85,B 0,C 180,E1 -498.454,E2 -498.454} C_VEL
LIN {X 0,Y 760.441,Z 303.319,A -85,B 0,C 180,E1 -500.69,E2 -500.69} C_VEL
LIN {X 0,Y 760.439,Z 303.317,A -85,B 0,C 180,E1 -503.26,E2 -503.26} C_VEL
LIN {X 0,Y 760.414,Z 303.315,A -85,B 0,C 180,E1 -505.813,E2 -505.813} C_VEL
LIN {X 0,Y 760.401,Z 303.317,A -85,B 0,C 180,E1 -507.937,E2 -507.937} C_VEL
LIN {X 0,Y 760.409,Z 303.317,A -85,B 0,C 180,E1 -509.983,E2 -509.983} C_VEL
LIN {X 0,Y 760.413,Z 303.32,A -85,B 0,C 180,E1 -512.165,E2 -512.165} C_VEL
LIN {X 0,Y 760.472,Z 303.321,A -85,B 0,C 180,E1 -514.508,E2 -514.508} C_VEL
LIN {X 0,Y 760.414,Z 303.325,A -85,B 0,C 180,E1 -515.633,E2 -515.633} C_VEL
LIN {X 0,Y 760.655,Z 310.006,A -85,B 0,C 180,E1 -516.242,E2 -516.242} C_VEL
LIN {X 0,Y 760.612,Z 338.897,A -85,B 0,C 180,E1 -518.811,E2 -518.811} C_VEL
LIN {X 0,Y 760.565,Z 367.516,A -85,B 0,C 180,E1 -521.312,E2 -521.312} C_VEL
LIN {X 0,Y 760.486,Z 395.077,A -85,B 0,C 180,E1 -523.685,E2 -523.685} C_VEL
LIN {X 0,Y 760.511,Z 420.76,A -85,B 0,C 180,E1 -525.873,E2 -525.873} C_VEL
LIN {X 0,Y 760.506,Z 439.666,A -85,B 0,C 180,E1 -527.47,E2 -527.47} C_VEL
LIN {X 0,Y 760.531,Z 578.391,A -85,B 0,C 180,E1 -528.798,E2 -528.798} C_VEL
LIN {X 0,Y 760.532,Z 593.043,A -85,B 0,C 180,E1 -529.05,E2 -529.05} C_VEL
LIN {X 0,Y 760.499,Z 607.539,A -85,B 0,C 180,E1 -529.419,E2 -529.419} C_VEL
LIN {X 0,Y 760.467,Z 620.359,A -85,B 0,C 180,E1 -529.854,E2 -529.854} C_VEL
LIN {X 0,Y 760.475,Z 632.943,A -85,B 0,C 180,E1 -530.396,E2 -530.396} C_VEL
LIN {X 0,Y 760.489,Z 644.22,A -85,B 0,C 180,E1 -530.992,E2 -530.992} C_VEL
LIN {X 0,Y 760.467,Z 654.691,A -85,B 0,C 180,E1 -531.659,E2 -531.659} C_VEL
LIN {X 0,Y 760.468,Z 665.1,A -85,B 0,C 180,E1 -532.458,E2 -532.458} C_VEL
LIN {X 0,Y 760.464,Z 673.691,A -85,B 0,C 180,E1 -533.256,E2 -533.256} C_VEL
LIN {X 0,Y 760.437,Z 681.922,A -85,B 0,C 180,E1 -534.185,E2 -534.185} C_VEL
LIN {X 0,Y 760.453,Z 687.673,A -85,B 0,C 180,E1 -534.98,E2 -534.98} C_VEL
LIN {X 0,Y 760.437,Z 692.404,A -85,B 0,C 180,E1 -535.774,E2 -535.774} C_VEL
LIN {X 0,Y 760.427,Z 697.305,A -85,B 0,C 180,E1 -536.832,E2 -536.832} C_VEL
LIN {X 0,Y 760.426,Z 700.729,A -85,B 0,C 180,E1 -537.889,E2 -537.889} C_VEL
LIN {X 0,Y 760.451,Z 702.77,A -85,B 0,C 180,E1 -538.945,E2 -538.945} C_VEL
LIN {X 0,Y 760.437,Z 703.493,A -85,B 0,C 180,E1 -540,E2 -540} C_VEL
LIN {X 0,Y 760.45,Z 702.898,A -85,B 0,C 180,E1 -541.056,E2 -541.056} C_VEL
LIN {X 0,Y 760.423,Z 700.971,A -85,B 0,C 180,E1 -542.112,E2 -542.112} C_VEL
LIN {X 0,Y 760.425,Z 697.663,A -85,B 0,C 180,E1 -543.168,E2 -543.168} C_VEL
LIN {X 0,Y 760.438,Z 692.884,A -85,B 0,C 180,E1 -544.226,E2 -544.226} C_VEL
LIN {X 0,Y 760.435,Z 686.478,A -85,B 0,C 180,E1 -545.285,E2 -545.285} C_VEL
LIN {X 0,Y 760.46,Z 679.351,A -85,B 0,C 180,E1 -546.213,E2 -546.213} C_VEL
LIN {X 0,Y 760.46,Z 670.542,A -85,B 0,C 180,E1 -547.143,E2 -547.143} C_VEL
LIN {X 0,Y 760.463,Z 663.74,A -85,B 0,C 180,E1 -547.744,E2 -547.744} C_VEL
LIN {X 0,Y 759.836,Z 659.765,A -85,B 0,C 180,E1 -548.068,E2 -548.068} C_VEL
LIN {X 0,Y 756.987,Z 653.097,A -85,B 0,C 180,E1 -548.581,E2 -548.581} C_VEL
LIN {X 0,Y 754.119,Z 646.108,A -85,B 0,C 180,E1 -549.065,E2 -549.065} C_VEL
LIN {X 0,Y 753.466,Z 641.455,A -85,B 0,C 180,E1 -549.343,E2 -549.343} C_VEL
LIN {X 0,Y 753.454,Z 629.247,A -85,B 0,C 180,E1 -549.961,E2 -549.961} C_VEL
LIN {X 0,Y 753.512,Z 615.486,A -85,B 0,C 180,E1 -550.511,E2 -550.511} C_VEL
LIN {X 0,Y 753.548,Z 602.361,A -85,B 0,C 180,E1 -550.917,E2 -550.917} C_VEL
LIN {X 0,Y 753.554,Z 588.191,A -85,B 0,C 180,E1 -551.24,E2 -551.24} C_VEL
LIN {X 0,Y 753.551,Z 573.044,A -85,B 0,C 180,E1 -551.46,E2 -551.46} C_VEL
LIN {X 0,Y 753.529,Z 440.099,A -85,B 0,C 180,E1 -552.732,E2 -552.732} C_VEL
LIN {X 0,Y 753.494,Z 439.586,A -85,B 0,C 180,E1 -552.746,E2 -552.746} C_VEL
LIN {X 0,Y 753.552,Z 410.572,A -85,B 0,C 180,E1 -555.224,E2 -555.224} C_VEL
LIN {X 0,Y 753.609,Z 381.666,A -85,B 0,C 180,E1 -557.722,E2 -557.722} C_VEL
LIN {X 0,Y 753.712,Z 352.92,A -85,B 0,C 180,E1 -560.239,E2 -560.239} C_VEL
LIN {X 0,Y 753.754,Z 323.849,A -85,B 0,C 180,E1 -562.829,E2 -562.829} C_VEL
LIN {X 0,Y 753.801,Z 306.384,A -85,B 0,C 180,E1 -564.407,E2 -564.407} C_VEL
LIN {X 0,Y 753.389,Z 304.195,A -85,B 0,C 180,E1 -564.628,E2 -564.628} C_VEL
LIN {X 0,Y 753.393,Z 304.191,A -85,B 0,C 180,E1 -566.807,E2 -566.807} C_VEL
LIN {X 0,Y 753.41,Z 304.193,A -85,B 0,C 180,E1 -569.083,E2 -569.083} C_VEL
LIN {X 0,Y 753.405,Z 304.201,A -85,B 0,C 180,E1 -571.375,E2 -571.375} C_VEL
LIN {X 0,Y 753.41,Z 304.189,A -85,B 0,C 180,E1 -573.905,E2 -573.905} C_VEL
LIN {X 0,Y 753.401,Z 304.189,A -85,B 0,C 180,E1 -576.016,E2 -576.016} C_VEL
LIN {X 0,Y 753.42,Z 304.187,A -85,B 0,C 180,E1 -577.85,E2 -577.85} C_VEL
LIN {X 0,Y 753.403,Z 304.189,A -85,B 0,C 180,E1 -579.904,E2 -579.904} C_VEL
LIN {X 0,Y 753.393,Z 304.19,A -85,B 0,C 180,E1 -582.021,E2 -582.021} C_VEL
LIN {X 0,Y 753.391,Z 304.192,A -85,B 0,C 180,E1 -584.284,E2 -584.284} C_VEL
LIN {X 0,Y 753.412,Z 304.194,A -85,B 0,C 180,E1 -586.53,E2 -586.53} C_VEL
LIN {X 0,Y 753.424,Z 304.196,A -85,B 0,C 180,E1 -588.855,E2 -588.855} C_VEL
LIN {X 0,Y 753.404,Z 304.189,A -85,B 0,C 180,E1 -591.471,E2 -591.471} C_VEL
LIN {X 0,Y 753.408,Z 304.19,A -85,B 0,C 180,E1 -593.983,E2 -593.983} C_VEL
LIN {X 0,Y 753.41,Z 304.192,A -85,B 0,C 180,E1 -596.095,E2 -596.095} C_VEL
LIN {X 0,Y 753.398,Z 304.197,A -85,B 0,C 180,E1 -598.625,E2 -598.625} C_VEL
LIN {X 0,Y 753.42,Z 304.187,A -85,B 0,C 180,E1 -601.09,E2 -601.09} C_VEL
LIN {X 0,Y 753.403,Z 304.189,A -85,B 0,C 180,E1 -603.496,E2 -603.496} C_VEL
LIN {X 0,Y 753.414,Z 304.194,A -85,B 0,C 180,E1 -605.854,E2 -605.854} C_VEL
LIN {X 0,Y 753.397,Z 304.195,A -85,B 0,C 180,E1 -608.391,E2 -608.391} C_VEL
LIN {X 0,Y 753.395,Z 304.193,A -85,B 0,C 180,E1 -610.446,E2 -610.446} C_VEL
LIN {X 0,Y 753.403,Z 304.189,A -85,B 0,C 180,E1 -612.692,E2 -612.692} C_VEL
LIN {X 0,Y 753.42,Z 304.188,A -85,B 0,C 180,E1 -615.213,E2 -615.213} C_VEL
LIN {X 0,Y 753.423,Z 304.198,A -85,B 0,C 180,E1 -617.653,E2 -617.653} C_VEL
LIN {X 0,Y 753.406,Z 304.197,A -85,B 0,C 180,E1 -619.826,E2 -619.826} C_VEL
LIN {X 0,Y 753.373,Z 304.194,A -85,B 0,C 180,E1 -622.252,E2 -622.252} C_VEL
LIN {X 0,Y 753.382,Z 304.192,A -85,B 0,C 180,E1 -622.437,E2 -622.437} C_VEL
LIN {X 0,Y 753.601,Z 310.482,A -85,B 0,C 180,E1 -622.506,E2 -622.506} C_VEL
LIN {X 0,Y 753.597,Z 433.571,A -85,B 0,C 180,E1 -623.697,E2 -623.697} C_VEL
LIN {X 0,Y 753.574,Z 447.641,A -85,B 0,C 180,E1 -623.938,E2 -623.938} C_VEL
LIN {X 0,Y 753.544,Z 462.475,A -85,B 0,C 180,E1 -624.317,E2 -624.317} C_VEL
LIN {X 0,Y 753.513,Z 476.424,A -85,B 0,C 180,E1 -624.8,E2 -624.8} C_VEL
LIN {X 0,Y 753.468,Z 488.563,A -85,B 0,C 180,E1 -625.334,E2 -625.334} C_VEL
LIN {X 0,Y 753.456,Z 499.705,A -85,B 0,C 180,E1 -625.935,E2 -625.935} C_VEL
LIN {X 0,Y 753.433,Z 509.039,A -85,B 0,C 180,E1 -626.536,E2 -626.536} C_VEL
LIN {X 0,Y 753.382,Z 519.467,A -85,B 0,C 180,E1 -627.336,E2 -627.336} C_VEL
LIN {X 0,Y 753.389,Z 528.106,A -85,B 0,C 180,E1 -628.135,E2 -628.135} C_VEL
LIN {X 0,Y 753.392,Z 536.424,A -85,B 0,C 180,E1 -629.068,E2 -629.068} C_VEL
LIN {X 0,Y 753.347,Z 543.132,A -85,B 0,C 180,E1 -630,E2 -630} C_VEL
LIN {X 0,Y 753.348,Z 549.107,A -85,B 0,C 180,E1 -631.066,E2 -631.066} C_VEL
LIN {X 0,Y 753.325,Z 553.511,A -85,B 0,C 180,E1 -632.132,E2 -632.132} C_VEL
LIN {X 0,Y 753.322,Z 556.495,A -85,B 0,C 180,E1 -633.198,E2 -633.198} C_VEL
LIN {X 0,Y 753.335,Z 558.118,A -85,B 0,C 180,E1 -634.266,E2 -634.266} C_VEL
LIN {X 0,Y 753.33,Z 558.423,A -85,B 0,C 180,E1 -635.335,E2 -635.335} C_VEL
LIN {X 0,Y 753.343,Z 557.408,A -85,B 0,C 180,E1 -636.406,E2 -636.406} C_VEL
LIN {X 0,Y 753.327,Z 555.043,A -85,B 0,C 180,E1 -637.48,E2 -637.48} C_VEL
LIN {X 0,Y 753.34,Z 551.249,A -85,B 0,C 180,E1 -638.556,E2 -638.556} C_VEL
LIN {X 0,Y 753.36,Z 547.364,A -85,B 0,C 180,E1 -639.364,E2 -639.364} C_VEL
LIN {X 0,Y 753.371,Z 542.558,A -85,B 0,C 180,E1 -640.175,E2 -640.175} C_VEL
LIN {X 0,Y 753.396,Z 535.582,A -85,B 0,C 180,E1 -641.123,E2 -641.123} C_VEL
LIN {X 0,Y 753.39,Z 528.267,A -85,B 0,C 180,E1 -641.939,E2 -641.939} C_VEL
LIN {X 0,Y 753.409,Z 519.337,A -85,B 0,C 180,E1 -642.765,E2 -642.765} C_VEL
LIN {X 0,Y 753.416,Z 510.676,A -85,B 0,C 180,E1 -643.44,E2 -643.44} C_VEL
LIN {X 0,Y 753.44,Z 500.214,A -85,B 0,C 180,E1 -644.125,E2 -644.125} C_VEL
LIN {X 0,Y 753.477,Z 489.504,A -85,B 0,C 180,E1 -644.71,E2 -644.71} C_VEL
LIN {X 0,Y 753.498,Z 478.059,A -85,B 0,C 180,E1 -645.225,E2 -645.225} C_VEL
LIN {X 0,Y 753.516,Z 464.622,A -85,B 0,C 180,E1 -645.708,E2 -645.708} C_VEL
LIN {X 0,Y 753.567,Z 449.754,A -85,B 0,C 180,E1 -646.105,E2 -646.105} C_VEL
LIN {X 0,Y 753.6,Z 435.629,A -85,B 0,C 180,E1 -646.364,E2 -646.364} C_VEL
LIN {X 0,Y 753.625,Z 412.757,A -85,B 0,C 180,E1 -646.607,E2 -646.607} C_VEL
LIN {X 0,Y 753.514,Z 305.052,A -85,B 0,C 180,E1 -647.637,E2 -647.637} C_VEL
LIN {X 0,Y 753.362,Z 304.194,A -85,B 0,C 180,E1 -647.658,E2 -647.658} C_VEL
LIN {X 0,Y 753.343,Z 304.196,A -85,B 0,C 180,E1 -649.556,E2 -649.556} C_VEL
LIN {X 0,Y 753.366,Z 304.195,A -85,B 0,C 180,E1 -651.833,E2 -651.833} C_VEL
LIN {X 0,Y 753.383,Z 304.202,A -85,B 0,C 180,E1 -654.336,E2 -654.336} C_VEL
LIN {X 0,Y 753.4,Z 304.193,A -85,B 0,C 180,E1 -656.807,E2 -656.807} C_VEL
LIN {X 0,Y 753.373,Z 304.193,A -85,B 0,C 180,E1 -659.077,E2 -659.077} C_VEL
LIN {X 0,Y 753.365,Z 304.193,A -85,B 0,C 180,E1 -661.377,E2 -661.377} C_VEL
LIN {X 0,Y 753.371,Z 304.197,A -85,B 0,C 180,E1 -663.907,E2 -663.907} C_VEL
LIN {X 0,Y 753.384,Z 304.197,A -85,B 0,C 180,E1 -666.515,E2 -666.515} C_VEL
LIN {X 0,Y 753.391,Z 304.193,A -85,B 0,C 180,E1 -668.65,E2 -668.65} C_VEL
LIN {X 0,Y 753.381,Z 304.191,A -85,B 0,C 180,E1 -671.309,E2 -671.309} C_VEL
LIN {X 0,Y 753.375,Z 304.194,A -85,B 0,C 180,E1 -673.514,E2 -673.514} C_VEL
LIN {X 0,Y 753.373,Z 304.199,A -85,B 0,C 180,E1 -675.788,E2 -675.788} C_VEL
LIN {X 0,Y 753.387,Z 304.203,A -85,B 0,C 180,E1 -678.055,E2 -678.055} C_VEL
LIN {X 0,Y 753.369,Z 304.195,A -85,B 0,C 180,E1 -680.507,E2 -680.507} C_VEL
LIN {X 0,Y 753.34,Z 304.195,A -85,B 0,C 180,E1 -682.817,E2 -682.817} C_VEL
LIN {X 0,Y 753.35,Z 304.194,A -85,B 0,C 180,E1 -684.906,E2 -684.906} C_VEL
LIN {X 0,Y 753.366,Z 304.192,A -85,B 0,C 180,E1 -686.802,E2 -686.802} C_VEL
LIN {X 0,Y 753.365,Z 304.192,A -85,B 0,C 180,E1 -688.802,E2 -688.802} C_VEL
LIN {X 0,Y 753.361,Z 304.193,A -85,B 0,C 180,E1 -690.924,E2 -690.924} C_VEL
LIN {X 0,Y 753.384,Z 304.193,A -85,B 0,C 180,E1 -693.195,E2 -693.195} C_VEL
LIN {X 0,Y 753.416,Z 304.196,A -85,B 0,C 180,E1 -695.854,E2 -695.854} C_VEL
LIN {X 0,Y 753.377,Z 304.192,A -85,B 0,C 180,E1 -698.395,E2 -698.395} C_VEL
LIN {X 0,Y 753.364,Z 304.193,A -85,B 0,C 180,E1 -700.445,E2 -700.445} C_VEL
LIN {X 0,Y 753.374,Z 304.192,A -85,B 0,C 180,E1 -702.691,E2 -702.691} C_VEL
LIN {X 0,Y 753.406,Z 304.194,A -85,B 0,C 180,E1 -705.216,E2 -705.216} C_VEL
LIN {X 0,Y 753.38,Z 304.192,A -85,B 0,C 180,E1 -706.44,E2 -706.44} C_VEL
LIN {X 0,Y 753.557,Z 325.379,A -85,B 0,C 180,E1 -706.648,E2 -706.648} C_VEL
LIN {X 0,Y 753.615,Z 433.208,A -85,B 0,C 180,E1 -707.69,E2 -707.69} C_VEL
LIN {X 0,Y 753.574,Z 447.159,A -85,B 0,C 180,E1 -707.928,E2 -707.928} C_VEL
LIN {X 0,Y 753.533,Z 460.783,A -85,B 0,C 180,E1 -708.268,E2 -708.268} C_VEL
LIN {X 0,Y 753.5,Z 473.156,A -85,B 0,C 180,E1 -708.675,E2 -708.675} C_VEL
LIN {X 0,Y 753.498,Z 486.118,A -85,B 0,C 180,E1 -709.217,E2 -709.217} C_VEL
LIN {X 0,Y 753.468,Z 497.848,A -85,B 0,C 180,E1 -709.826,E2 -709.826} C_VEL
LIN {X 0,Y 753.421,Z 508.571,A -85,B 0,C 180,E1 -710.501,E2 -710.501} C_VEL
LIN {X 0,Y 753.405,Z 519.187,A -85,B 0,C 180,E1 -711.31,E2 -711.31} C_VEL
LIN {X 0,Y 753.392,Z 527.948,A -85,B 0,C 180,E1 -712.118,E2 -712.118} C_VEL
LIN {X 0,Y 753.377,Z 536.343,A -85,B 0,C 180,E1 -713.058,E2 -713.058} C_VEL
LIN {X 0,Y 753.371,Z 542.199,A -85,B 0,C 180,E1 -713.862,E2 -713.862} C_VEL
LIN {X 0,Y 753.36,Z 548.447,A -85,B 0,C 180,E1 -714.932,E2 -714.932} C_VEL
LIN {X 0,Y 753.339,Z 552.029,A -85,B 0,C 180,E1 -715.734,E2 -715.734} C_VEL
LIN {X 0,Y 753.323,Z 555.546,A -85,B 0,C 180,E1 -716.802,E2 -716.802} C_VEL
LIN {X 0,Y 753.317,Z 557.672,A -85,B 0,C 180,E1 -717.868,E2 -717.868} C_VEL
LIN {X 0,Y 753.349,Z 558.474,A -85,B 0,C 180,E1 -718.934,E2 -718.934} C_VEL
LIN {X 0,Y 753.339,Z 557.968,A -85,B 0,C 180,E1 -720,E2 -720} C_VEL
LIN {X 0,Y 753.352,Z 556.136,A -85,B 0,C 180,E1 -721.065,E2 -721.065} C_VEL
LIN {X 0,Y 753.328,Z 552.914,A -85,B 0,C 180,E1 -722.131,E2 -722.131} C_VEL
LIN {X 0,Y 753.358,Z 548.24,A -85,B 0,C 180,E1 -723.198,E2 -723.198} C_VEL
LIN {X 0,Y 753.344,Z 541.947,A -85,B 0,C 180,E1 -724.266,E2 -724.266} C_VEL
LIN {X 0,Y 753.374,Z 534.945,A -85,B 0,C 180,E1 -725.201,E2 -725.201} C_VEL
LIN {X 0,Y 753.377,Z 526.279,A -85,B 0,C 180,E1 -726.138,E2 -726.138} C_VEL
LIN {X 0,Y 753.427,Z 517.231,A -85,B 0,C 180,E1 -726.942,E2 -726.942} C_VEL
LIN {X 0,Y 753.432,Z 506.232,A -85,B 0,C 180,E1 -727.747,E2 -727.747} C_VEL
LIN {X 0,Y 753.46,Z 495.081,A -85,B 0,C 180,E1 -728.419,E2 -728.419} C_VEL
LIN {X 0,Y 753.512,Z 482.769,A -85,B 0,C 180,E1 -729.025,E2 -729.025} C_VEL
LIN {X 0,Y 753.537,Z 468.964,A -85,B 0,C 180,E1 -729.564,E2 -729.564} C_VEL
LIN {X 0,Y 753.558,Z 454.92,A -85,B 0,C 180,E1 -729.982,E2 -729.982} C_VEL
LIN {X 0,Y 753.561,Z 440.435,A -85,B 0,C 180,E1 -730.29,E2 -730.29} C_VEL
LIN {X 0,Y 753.603,Z 426.524,A -85,B 0,C 180,E1 -730.476,E2 -730.476} C_VEL
LIN {X 0,Y 753.594,Z 305.113,A -85,B 0,C 180,E1 -731.635,E2 -731.635} C_VEL
LIN {X 0,Y 753.424,Z 304.187,A -85,B 0,C 180,E1 -731.649,E2 -731.649} C_VEL
LIN {X 0,Y 753.388,Z 304.195,A -85,B 0,C 180,E1 -733.988,E2 -733.988} C_VEL
LIN {X 0,Y 753.397,Z 304.199,A -85,B 0,C 180,E1 -736.195,E2 -736.195} C_VEL
LIN {X 0,Y 753.433,Z 304.192,A -85,B 0,C 180,E1 -738.51,E2 -738.51} C_VEL
LIN {X 0,Y 753.421,Z 304.189,A -85,B 0,C 180,E1 -740.688,E2 -740.688} C_VEL
LIN {X 0,Y 753.404,Z 304.189,A -85,B 0,C 180,E1 -743.013,E2 -743.013} C_VEL
LIN {X 0,Y 753.431,Z 304.191,A -85,B 0,C 180,E1 -745.606,E2 -745.606} C_VEL
LIN {X 0,Y 753.407,Z 304.192,A -85,B 0,C 180,E1 -748.304,E2 -748.304} C_VEL
LIN {X 0,Y 753.415,Z 304.187,A -85,B 0,C 180,E1 -750.752,E2 -750.752} C_VEL
LIN {X 0,Y 753.422,Z 304.192,A -85,B 0,C 180,E1 -753.265,E2 -753.265} C_VEL
LIN {X 0,Y 753.396,Z 304.195,A -85,B 0,C 180,E1 -755.854,E2 -755.854} C_VEL
LIN {X 0,Y 753.412,Z 304.191,A -85,B 0,C 180,E1 -757.85,E2 -757.85} C_VEL
LIN {X 0,Y 753.379,Z 304.194,A -85,B 0,C 180,E1 -759.905,E2 -759.905} C_VEL
LIN {X 0,Y 753.372,Z 304.193,A -85,B 0,C 180,E1 -762.022,E2 -762.022} C_VEL
LIN {X 0,Y 753.367,Z 304.193,A -85,B 0,C 180,E1 -764.282,E2 -764.282} C_VEL
LIN {X 0,Y 753.402,Z 304.192,A -85,B 0,C 180,E1 -766.529,E2 -766.529} C_VEL
LIN {X 0,Y 753.415,Z 304.198,A -85,B 0,C 180,E1 -768.855,E2 -768.855} C_VEL
LIN {X 0,Y 753.376,Z 304.195,A -85,B 0,C 180,E1 -771.351,E2 -771.351} C_VEL
LIN {X 0,Y 753.35,Z 304.196,A -85,B 0,C 180,E1 -773.483,E2 -773.483} C_VEL
LIN {X 0,Y 753.38,Z 304.192,A -85,B 0,C 180,E1 -775.839,E2 -775.839} C_VEL
LIN {X 0,Y 753.351,Z 304.198,A -85,B 0,C 180,E1 -777.996,E2 -777.996} C_VEL
LIN {X 0,Y 753.384,Z 304.203,A -85,B 0,C 180,E1 -780.478,E2 -780.478} C_VEL
LIN {X 0,Y 753.367,Z 304.196,A -85,B 0,C 180,E1 -782.898,E2 -782.898} C_VEL
LIN {X 0,Y 753.356,Z 304.258,A -85,B 0,C 180,E1 -785.212,E2 -785.212} C_VEL
LIN {X 0,Y 753.844,Z 307.167,A -85,B 0,C 180,E1 -785.489,E2 -785.489} C_VEL
LIN {X 0,Y 753.791,Z 334.296,A -85,B 0,C 180,E1 -787.893,E2 -787.893} C_VEL
LIN {X 0,Y 753.688,Z 363.722,A -85,B 0,C 180,E1 -790.454,E2 -790.454} C_VEL
LIN {X 0,Y 753.566,Z 391.676,A -85,B 0,C 180,E1 -792.849,E2 -792.849} C_VEL
LIN {X 0,Y 753.474,Z 417.716,A -85,B 0,C 180,E1 -795.054,E2 -795.054} C_VEL
LIN {X 0,Y 753.45,Z 442.189,A -85,B 0,C 180,E1 -797.108,E2 -797.108} C_VEL
LIN {X 0,Y 753.478,Z 444.65,A -85,B 0,C 180,E1 -797.308,E2 -797.308} C_VEL
LIN {X 0,Y 753.545,Z 583.002,A -85,B 0,C 180,E1 -798.642,E2 -798.642} C_VEL
LIN {X 0,Y 753.551,Z 597.784,A -85,B 0,C 180,E1 -798.896,E2 -798.896} C_VEL
LIN {X 0,Y 753.539,Z 611.79,A -85,B 0,C 180,E1 -799.252,E2 -799.252} C_VEL
LIN {X 0,Y 753.48,Z 624.784,A -85,B 0,C 180,E1 -799.691,E2 -799.691} C_VEL
LIN {X 0,Y 753.475,Z 637.536,A -85,B 0,C 180,E1 -800.24,E2 -800.24} C_VEL
LIN {X 0,Y 753.449,Z 649.999,A -85,B 0,C 180,E1 -800.907,E2 -800.907} C_VEL
LIN {X 0,Y 753.413,Z 660.339,A -85,B 0,C 180,E1 -801.58,E2 -801.58} C_VEL
LIN {X 0,Y 753.401,Z 670.636,A -85,B 0,C 180,E1 -802.387,E2 -802.387} C_VEL
LIN {X 0,Y 753.389,Z 679.136,A -85,B 0,C 180,E1 -803.192,E2 -803.192} C_VEL
LIN {X 0,Y 753.387,Z 687.263,A -85,B 0,C 180,E1 -804.13,E2 -804.13} C_VEL
LIN {X 0,Y 753.376,Z 692.979,A -85,B 0,C 180,E1 -804.933,E2 -804.933} C_VEL
LIN {X 0,Y 753.34,Z 697.643,A -85,B 0,C 180,E1 -805.734,E2 -805.734} C_VEL
LIN {X 0,Y 753.354,Z 702.484,A -85,B 0,C 180,E1 -806.802,E2 -806.802} C_VEL
LIN {X 0,Y 753.325,Z 705.85,A -85,B 0,C 180,E1 -807.868,E2 -807.868} C_VEL
LIN {X 0,Y 753.345,Z 707.836,A -85,B 0,C 180,E1 -808.934,E2 -808.934} C_VEL
LIN {X 0,Y 753.339,Z 708.5,A -85,B 0,C 180,E1 -810,E2 -810} C_VEL
LIN {X 0,Y 753.345,Z 707.836,A -85,B 0,C 180,E1 -811.065,E2 -811.065} C_VEL
LIN {X 0,Y 753.325,Z 705.85,A -85,B 0,C 180,E1 -812.131,E2 -812.131} C_VEL
LIN {X 0,Y 753.354,Z 702.484,A -85,B 0,C 180,E1 -813.198,E2 -813.198} C_VEL
LIN {X 0,Y 753.338,Z 697.644,A -85,B 0,C 180,E1 -814.266,E2 -814.266} C_VEL
LIN {X 0,Y 753.357,Z 691.174,A -85,B 0,C 180,E1 -815.335,E2 -815.335} C_VEL
LIN {X 0,Y 753.398,Z 683.975,A -85,B 0,C 180,E1 -816.272,E2 -816.272} C_VEL
LIN {X 0,Y 753.393,Z 675.082,A -85,B 0,C 180,E1 -817.21,E2 -817.21} C_VEL
LIN {X 0,Y 753.412,Z 665.748,A -85,B 0,C 180,E1 -818.016,E2 -818.016} C_VEL
LIN {X 0,Y 753.435,Z 654.353,A -85,B 0,C 180,E1 -818.824,E2 -818.824} C_VEL
LIN {X 0,Y 753.463,Z 642.757,A -85,B 0,C 180,E1 -819.498,E2 -819.498} C_VEL
LIN {X 0,Y 753.501,Z 629.783,A -85,B 0,C 180,E1 -820.109,E2 -820.109} C_VEL
LIN {X 0,Y 753.514,Z 616.237,A -85,B 0,C 180,E1 -820.613,E2 -820.613} C_VEL
LIN {X 0,Y 753.567,Z 602.337,A -85,B 0,C 180,E1 -821.002,E2 -821.002} C_VEL
LIN {X 0,Y 753.57,Z 588.745,A -85,B 0,C 180,E1 -821.273,E2 -821.273} C_VEL
LIN {X 0,Y 753.566,Z 573.562,A -85,B 0,C 180,E1 -821.46,E2 -821.46} C_VEL
LIN {X 0,Y 753.583,Z 445.348,A -85,B 0,C 180,E1 -822.684,E2 -822.684} C_VEL
LIN {X 0,Y 753.468,Z 444.484,A -85,B 0,C 180,E1 -822.7,E2 -822.7} C_VEL
LIN {X 0,Y 753.474,Z 419.397,A -85,B 0,C 180,E1 -824.804,E2 -824.804} C_VEL
LIN {X 0,Y 753.547,Z 394.949,A -85,B 0,C 180,E1 -826.873,E2 -826.873} C_VEL
LIN {X 0,Y 753.651,Z 366.993,A -85,B 0,C 180,E1 -829.265,E2 -829.265} C_VEL
LIN {X 0,Y 753.75,Z 339.211,A -85,B 0,C 180,E1 -831.677,E2 -831.677} C_VEL
LIN {X 0,Y 753.848,Z 311.412,A -85,B 0,C 180,E1 -834.131,E2 -834.131} C_VEL
LIN {X 0,Y 753.753,Z 306.023,A -85,B 0,C 180,E1 -834.616,E2 -834.616} C_VEL
LIN {X 0,Y 753.35,Z 304.2,A -85,B 0,C 180,E1 -834.807,E2 -834.807} C_VEL
LIN {X 0,Y 753.371,Z 304.193,A -85,B 0,C 180,E1 -836.804,E2 -836.804} C_VEL
LIN {X 0,Y 753.387,Z 304.193,A -85,B 0,C 180,E1 -839.08,E2 -839.08} C_VEL
LIN {X 0,Y 753.376,Z 304.201,A -85,B 0,C 180,E1 -841.376,E2 -841.376} C_VEL
LIN {X 0,Y 753.365,Z 304.197,A -85,B 0,C 180,E1 -843.907,E2 -843.907} C_VEL
LIN {X 0,Y 753.354,Z 304.196,A -85,B 0,C 180,E1 -846.012,E2 -846.012} C_VEL
LIN {X 0,Y 753.36,Z 304.197,A -85,B 0,C 180,E1 -847.853,E2 -847.853} C_VEL
LIN {X 0,Y 753.347,Z 304.197,A -85,B 0,C 180,E1 -849.907,E2 -849.907} C_VEL
LIN {X 0,Y 753.352,Z 304.195,A -85,B 0,C 180,E1 -852.024,E2 -852.024} C_VEL
LIN {X 0,Y 753.329,Z 304.198,A -85,B 0,C 180,E1 -854.279,E2 -854.279} C_VEL
LIN {X 0,Y 753.386,Z 304.193,A -85,B 0,C 180,E1 -856.528,E2 -856.528} C_VEL
LIN {X 0,Y 753.413,Z 304.197,A -85,B 0,C 180,E1 -858.856,E2 -858.856} C_VEL
LIN {X 0,Y 753.37,Z 304.195,A -85,B 0,C 180,E1 -861.47,E2 -861.47} C_VEL
LIN {X 0,Y 753.373,Z 304.194,A -85,B 0,C 180,E1 -863.485,E2 -863.485} C_VEL
LIN {X 0,Y 753.388,Z 304.19,A -85,B 0,C 180,E1 -865.838,E2 -865.838} C_VEL
LIN {X 0,Y 753.359,Z 304.195,A -85,B 0,C 180,E1 -867.997,E2 -867.997} C_VEL
LIN {X 0,Y 753.375,Z 304.193,A -85,B 0,C 180,E1 -869.864,E2 -869.864} C_VEL
LIN {X 0,Y 753.368,Z 304.196,A -85,B 0,C 180,E1 -872.039,E2 -872.039} C_VEL
LIN {X 0,Y 753.438,Z 304.195,A -85,B 0,C 180,E1 -874.393,E2 -874.393} C_VEL
LIN {X 0,Y 753.388,Z 304.268,A -85,B 0,C 180,E1 -875.476,E2 -875.476} C_VEL
LIN {X 0,Y 753.817,Z 308.407,A -85,B 0,C 180,E1 -875.868,E2 -875.868} C_VEL
LIN {X 0,Y 753.785,Z 334.087,A -85,B 0,C 180,E1 -878.18,E2 -878.18} C_VEL
LIN {X 0,Y 753.656,Z 364.584,A -85,B 0,C 180,E1 -880.876,E2 -880.876} C_VEL
LIN {X 0,Y 753.552,Z 395.082,A -85,B 0,C 180,E1 -883.531,E2 -883.531} C_VEL
LIN {X 0,Y 753.523,Z 422.37,A -85,B 0,C 180,E1 -885.877,E2 -885.877} C_VEL
LIN {X 0,Y 753.501,Z 439.608,A -85,B 0,C 180,E1 -887.346,E2 -887.346} C_VEL
LIN {X 0,Y 753.6,Z 512.154,A -85,B 0,C 180,E1 -888.048,E2 -888.048} C_VEL
LIN {X 0,Y 753.569,Z 578.382,A -85,B 0,C 180,E1 -888.693,E2 -888.693} C_VEL
LIN {X 0,Y 753.575,Z 592.293,A -85,B 0,C 180,E1 -888.931,E2 -888.931} C_VEL
LIN {X 0,Y 753.525,Z 606.442,A -85,B 0,C 180,E1 -889.286,E2 -889.286} C_VEL
LIN {X 0,Y 753.471,Z 620.372,A -85,B 0,C 180,E1 -889.759,E2 -889.759} C_VEL
LIN {X 0,Y 753.456,Z 632.482,A -85,B 0,C 180,E1 -890.283,E2 -890.283} C_VEL
LIN {X 0,Y 753.449,Z 644.226,A -85,B 0,C 180,E1 -890.907,E2 -890.907} C_VEL
LIN {X 0,Y 753.414,Z 654.7,A -85,B 0,C 180,E1 -891.58,E2 -891.58} C_VEL
LIN {X 0,Y 753.402,Z 665.108,A -85,B 0,C 180,E1 -892.387,E2 -892.387} C_VEL
LIN {X 0,Y 753.39,Z 673.691,A -85,B 0,C 180,E1 -893.192,E2 -893.192} C_VEL
LIN {X 0,Y 753.359,Z 682.317,A -85,B 0,C 180,E1 -894.181,E2 -894.181} C_VEL
LIN {X 0,Y 753.361,Z 689.355,A -85,B 0,C 180,E1 -895.2,E2 -895.2} C_VEL
LIN {X 0,Y 753.364,Z 695.044,A -85,B 0,C 180,E1 -896.269,E2 -896.269} C_VEL
LIN {X 0,Y 753.333,Z 699.195,A -85,B 0,C 180,E1 -897.336,E2 -897.336} C_VEL
LIN {X 0,Y 753.341,Z 701.92,A -85,B 0,C 180,E1 -898.402,E2 -898.402} C_VEL
LIN {X 0,Y 753.34,Z 703.297,A -85,B 0,C 180,E1 -899.467,E2 -899.467} C_VEL
LIN {X 0,Y 753.338,Z 703.359,A -85,B 0,C 180,E1 -900.533,E2 -900.533} C_VEL
LIN {X 0,Y 753.334,Z 702.099,A -85,B 0,C 180,E1 -901.599,E2 -901.599} C_VEL
LIN {X 0,Y 753.332,Z 699.492,A -85,B 0,C 180,E1 -902.665,E2 -902.665} C_VEL
LIN {X 0,Y 753.365,Z 695.458,A -85,B 0,C 180,E1 -903.732,E2 -903.732} C_VEL
LIN {X 0,Y 753.36,Z 689.895,A -85,B 0,C 180,E1 -904.8,E2 -904.8} C_VEL
LIN {X 0,Y 753.349,Z 682.647,A -85,B 0,C 180,E1 -905.865,E2 -905.865} C_VEL
LIN {X 0,Y 753.39,Z 674.554,A -85,B 0,C 180,E1 -906.808,E2 -906.808} C_VEL
LIN {X 0,Y 753.401,Z 666.13,A -85,B 0,C 180,E1 -907.613,E2 -907.613} C_VEL
LIN {X 0,Y 753.412,Z 655.988,A -85,B 0,C 180,E1 -908.42,E2 -908.42} C_VEL
LIN {X 0,Y 753.454,Z 644.609,A -85,B 0,C 180,E1 -909.161,E2 -909.161} C_VEL
LIN {X 0,Y 753.466,Z 641.455,A -85,B 0,C 180,E1 -909.343,E2 -909.343} C_VEL
LIN {X 0,Y 752.832,Z 636.736,A -85,B 0,C 180,E1 -909.61,E2 -909.61} C_VEL
LIN {X 0,Y 750.036,Z 628.953,A -85,B 0,C 180,E1 -910.027,E2 -910.027} C_VEL
LIN {X 0,Y 747.205,Z 620.836,A -85,B 0,C 180,E1 -910.405,E2 -910.405} C_VEL
LIN {X 0,Y 746.512,Z 615.597,A -85,B 0,C 180,E1 -910.607,E2 -910.607} C_VEL
LIN {X 0,Y 746.577,Z 602.336,A -85,B 0,C 180,E1 -911.021,E2 -911.021} C_VEL
LIN {X 0,Y 746.604,Z 588.175,A -85,B 0,C 180,E1 -911.346,E2 -911.346} C_VEL
LIN {X 0,Y 746.612,Z 573.027,A -85,B 0,C 180,E1 -911.568,E2 -911.568} C_VEL
LIN {X 0,Y 746.631,Z 440.853,A -85,B 0,C 180,E1 -912.844,E2 -912.844} C_VEL
LIN {X 0,Y 746.481,Z 439.553,A -85,B 0,C 180,E1 -912.87,E2 -912.87} C_VEL
LIN {X 0,Y 746.587,Z 408.961,A -85,B 0,C 180,E1 -915.509,E2 -915.509} C_VEL
LIN {X 0,Y 746.66,Z 381.661,A -85,B 0,C 180,E1 -917.893,E2 -917.893} C_VEL
LIN {X 0,Y 746.82,Z 352.753,A -85,B 0,C 180,E1 -920.449,E2 -920.449} C_VEL
LIN {X 0,Y 746.934,Z 323.125,A -85,B 0,C 180,E1 -923.114,E2 -923.114} C_VEL
LIN {X 0,Y 747.063,Z 309.389,A -85,B 0,C 180,E1 -924.365,E2 -924.365} C_VEL
LIN {X 0,Y 746.323,Z 305.077,A -85,B 0,C 180,E1 -924.797,E2 -924.797} C_VEL
LIN {X 0,Y 746.36,Z 305.069,A -85,B 0,C 180,E1 -926.93,E2 -926.93} C_VEL
LIN {X 0,Y 746.368,Z 305.073,A -85,B 0,C 180,E1 -929.217,E2 -929.217} C_VEL
LIN {X 0,Y 746.374,Z 305.069,A -85,B 0,C 180,E1 -931.705,E2 -931.705} C_VEL
LIN {X 0,Y 746.372,Z 305.064,A -85,B 0,C 180,E1 -934.325,E2 -934.325} C_VEL
LIN {X 0,Y 746.355,Z 305.066,A -85,B 0,C 180,E1 -936.246,E2 -936.246} C_VEL
LIN {X 0,Y 746.375,Z 305.071,A -85,B 0,C 180,E1 -938.838,E2 -938.838} C_VEL
LIN {X 0,Y 746.401,Z 305.066,A -85,B 0,C 180,E1 -941.345,E2 -941.345} C_VEL
LIN {X 0,Y 746.357,Z 305.066,A -85,B 0,C 180,E1 -943.986,E2 -943.986} C_VEL
LIN {X 0,Y 746.361,Z 305.068,A -85,B 0,C 180,E1 -946.272,E2 -946.272} C_VEL
LIN {X 0,Y 746.399,Z 305.069,A -85,B 0,C 180,E1 -948.936,E2 -948.936} C_VEL
LIN {X 0,Y 746.379,Z 305.067,A -85,B 0,C 180,E1 -951.162,E2 -951.162} C_VEL
LIN {X 0,Y 746.362,Z 305.066,A -85,B 0,C 180,E1 -953.813,E2 -953.813} C_VEL
LIN {X 0,Y 746.361,Z 305.076,A -85,B 0,C 180,E1 -956.379,E2 -956.379} C_VEL
LIN {X 0,Y 746.352,Z 305.074,A -85,B 0,C 180,E1 -958.653,E2 -958.653} C_VEL
LIN {X 0,Y 746.369,Z 305.068,A -85,B 0,C 180,E1 -960.79,E2 -960.79} C_VEL
LIN {X 0,Y 746.37,Z 305.064,A -85,B 0,C 180,E1 -963.226,E2 -963.226} C_VEL
LIN {X 0,Y 746.371,Z 305.067,A -85,B 0,C 180,E1 -965.611,E2 -965.611} C_VEL
LIN {X 0,Y 746.369,Z 305.072,A -85,B 0,C 180,E1 -968.293,E2 -968.293} C_VEL
LIN {X 0,Y 746.354,Z 305.073,A -85,B 0,C 180,E1 -970.254,E2 -970.254} C_VEL
LIN {X 0,Y 746.366,Z 305.067,A -85,B 0,C 180,E1 -972.524,E2 -972.524} C_VEL
LIN {X 0,Y 746.379,Z 305.065,A -85,B 0,C 180,E1 -975.154,E2 -975.154} C_VEL
LIN {X 0,Y 746.38,Z 305.072,A -85,B 0,C 180,E1 -977.535,E2 -977.535} C_VEL
LIN {X 0,Y 746.373,Z 305.067,A -85,B 0,C 180,E1 -980.195,E2 -980.195} C_VEL
LIN {X 0,Y 746.343,Z 305.196,A -85,B 0,C 180,E1 -982.331,E2 -982.331} C_VEL
LIN {X 0,Y 746.673,Z 308.468,A -85,B 0,C 180,E1 -982.369,E2 -982.369} C_VEL
LIN {X 0,Y 746.647,Z 433.275,A -85,B 0,C 180,E1 -983.587,E2 -983.587} C_VEL
LIN {X 0,Y 746.614,Z 446.285,A -85,B 0,C 180,E1 -983.807,E2 -983.807} C_VEL
LIN {X 0,Y 746.538,Z 459.403,A -85,B 0,C 180,E1 -984.125,E2 -984.125} C_VEL
LIN {X 0,Y 746.536,Z 473.084,A -85,B 0,C 180,E1 -984.572,E2 -984.572} C_VEL
LIN {X 0,Y 746.461,Z 486.776,A -85,B 0,C 180,E1 -985.156,E2 -985.156} C_VEL
LIN {X 0,Y 746.44,Z 498.228,A -85,B 0,C 180,E1 -985.762,E2 -985.762} C_VEL
LIN {X 0,Y 746.368,Z 507.803,A -85,B 0,C 180,E1 -986.368,E2 -986.368} C_VEL
LIN {X 0,Y 746.36,Z 516.814,A -85,B 0,C 180,E1 -987.041,E2 -987.041} C_VEL
LIN {X 0,Y 746.302,Z 525.883,A -85,B 0,C 180,E1 -987.849,E2 -987.849} C_VEL
LIN {X 0,Y 746.302,Z 533.466,A -85,B 0,C 180,E1 -988.656,E2 -988.656} C_VEL
LIN {X 0,Y 746.279,Z 539.797,A -85,B 0,C 180,E1 -989.462,E2 -989.462} C_VEL
LIN {X 0,Y 746.286,Z 545.037,A -85,B 0,C 180,E1 -990.269,E2 -990.269} C_VEL
LIN {X 0,Y 746.251,Z 549.321,A -85,B 0,C 180,E1 -991.076,E2 -991.076} C_VEL
LIN {X 0,Y 746.242,Z 551.7,A -85,B 0,C 180,E1 -991.614,E2 -991.614} C_VEL
LIN {X 0,Y 746.245,Z 555.319,A -85,B 0,C 180,E1 -992.69,E2 -992.69} C_VEL
LIN {X 0,Y 746.284,Z 557.549,A -85,B 0,C 180,E1 -993.767,E2 -993.767} C_VEL
LIN {X 0,Y 746.259,Z 558.451,A -85,B 0,C 180,E1 -994.846,E2 -994.846} C_VEL
LIN {X 0,Y 746.267,Z 558.033,A -85,B 0,C 180,E1 -995.926,E2 -995.926} C_VEL
LIN {X 0,Y 746.262,Z 556.277,A -85,B 0,C 180,E1 -997.009,E2 -997.009} C_VEL
LIN {X 0,Y 746.241,Z 553.146,A -85,B 0,C 180,E1 -998.094,E2 -998.094} C_VEL
LIN {X 0,Y 746.267,Z 548.54,A -85,B 0,C 180,E1 -999.182,E2 -999.182} C_VEL
LIN {X 0,Y 746.292,Z 542.232,A -85,B 0,C 180,E1 -1000.272,E2 -1000.272} C_VEL
LIN {X 0,Y 746.293,Z 535.173,A -85,B 0,C 180,E1 -1001.23,E2 -1001.23} C_VEL
LIN {X 0,Y 746.312,Z 527.766,A -85,B 0,C 180,E1 -1002.054,E2 -1002.054} C_VEL
LIN {X 0,Y 746.36,Z 518.996,A -85,B 0,C 180,E1 -1002.866,E2 -1002.866} C_VEL
LIN {X 0,Y 746.368,Z 509.965,A -85,B 0,C 180,E1 -1003.569,E2 -1003.569} C_VEL
LIN {X 0,Y 746.408,Z 499.37,A -85,B 0,C 180,E1 -1004.261,E2 -1004.261} C_VEL
LIN {X 0,Y 746.469,Z 488.051,A -85,B 0,C 180,E1 -1004.873,E2 -1004.873} C_VEL
LIN {X 0,Y 746.505,Z 475.061,A -85,B 0,C 180,E1 -1005.441,E2 -1005.441} C_VEL
LIN {X 0,Y 746.565,Z 460.719,A -85,B 0,C 180,E1 -1005.928,E2 -1005.928} C_VEL
LIN {X 0,Y 746.59,Z 446.605,A -85,B 0,C 180,E1 -1006.277,E2 -1006.277} C_VEL
LIN {X 0,Y 746.63,Z 433.281,A -85,B 0,C 180,E1 -1006.503,E2 -1006.503} C_VEL
LIN {X 0,Y 746.488,Z 305.931,A -85,B 0,C 180,E1 -1007.749,E2 -1007.749} C_VEL
LIN {X 0,Y 746.319,Z 305.073,A -85,B 0,C 180,E1 -1007.777,E2 -1007.777} C_VEL
LIN {X 0,Y 746.355,Z 305.076,A -85,B 0,C 180,E1 -1010.319,E2 -1010.319} C_VEL
LIN {X 0,Y 746.335,Z 305.079,A -85,B 0,C 180,E1 -1012.631,E2 -1012.631} C_VEL
LIN {X 0,Y 746.306,Z 305.075,A -85,B 0,C 180,E1 -1014.983,E2 -1014.983} C_VEL
LIN {X 0,Y 746.317,Z 305.071,A -85,B 0,C 180,E1 -1017.38,E2 -1017.38} C_VEL
LIN {X 0,Y 746.34,Z 305.071,A -85,B 0,C 180,E1 -1019.829,E2 -1019.829} C_VEL
LIN {X 0,Y 746.363,Z 305.077,A -85,B 0,C 180,E1 -1022.367,E2 -1022.367} C_VEL
LIN {X 0,Y 746.327,Z 305.071,A -85,B 0,C 180,E1 -1024.925,E2 -1024.925} C_VEL
LIN {X 0,Y 746.318,Z 305.071,A -85,B 0,C 180,E1 -1027.083,E2 -1027.083} C_VEL
LIN {X 0,Y 746.341,Z 305.068,A -85,B 0,C 180,E1 -1028.962,E2 -1028.962} C_VEL
LIN {X 0,Y 746.36,Z 305.066,A -85,B 0,C 180,E1 -1031.341,E2 -1031.341} C_VEL
LIN {X 0,Y 746.335,Z 305.079,A -85,B 0,C 180,E1 -1033.988,E2 -1033.988} C_VEL
LIN {X 0,Y 746.355,Z 305.074,A -85,B 0,C 180,E1 -1036.273,E2 -1036.273} C_VEL
LIN {X 0,Y 746.338,Z 305.068,A -85,B 0,C 180,E1 -1038.932,E2 -1038.932} C_VEL
LIN {X 0,Y 746.306,Z 305.072,A -85,B 0,C 180,E1 -1041.169,E2 -1041.169} C_VEL
LIN {X 0,Y 746.315,Z 305.069,A -85,B 0,C 180,E1 -1043.082,E2 -1043.082} C_VEL
LIN {X 0,Y 746.354,Z 305.075,A -85,B 0,C 180,E1 -1045.73,E2 -1045.73} C_VEL
LIN {X 0,Y 746.36,Z 305.069,A -85,B 0,C 180,E1 -1048.295,E2 -1048.295} C_VEL
LIN {X 0,Y 746.331,Z 305.069,A -85,B 0,C 180,E1 -1050.789,E2 -1050.789} C_VEL
LIN {X 0,Y 746.343,Z 305.07,A -85,B 0,C 180,E1 -1053.225,E2 -1053.225} C_VEL
LIN {X 0,Y 746.365,Z 305.075,A -85,B 0,C 180,E1 -1055.611,E2 -1055.611} C_VEL
LIN {X 0,Y 746.352,Z 305.068,A -85,B 0,C 180,E1 -1058.297,E2 -1058.297} C_VEL
LIN {X 0,Y 746.322,Z 305.072,A -85,B 0,C 180,E1 -1060.253,E2 -1060.253} C_VEL
LIN {X 0,Y 746.343,Z 305.068,A -85,B 0,C 180,E1 -1062.523,E2 -1062.523} C_VEL
LIN {X 0,Y 746.368,Z 305.07,A -85,B 0,C 180,E1 -1065.157,E2 -1065.157} C_VEL
LIN {X 0,Y 746.367,Z 305.26,A -85,B 0,C 180,E1 -1066.332,E2 -1066.332} C_VEL
LIN {X 0,Y 746.636,Z 308.307,A -85,B 0,C 180,E1 -1066.367,E2 -1066.367} C_VEL
LIN {X 0,Y 746.656,Z 433.747,A -85,B 0,C 180,E1 -1067.591,E2 -1067.591} C_VEL
LIN {X 0,Y 746.6,Z 448.252,A -85,B 0,C 180,E1 -1067.848,E2 -1067.848} C_VEL
LIN {X 0,Y 746.547,Z 461.581,A -85,B 0,C 180,E1 -1068.191,E2 -1068.191} C_VEL
LIN {X 0,Y 746.502,Z 472.887,A -85,B 0,C 180,E1 -1068.567,E2 -1068.567} C_VEL
LIN {X 0,Y 746.482,Z 484.436,A -85,B 0,C 180,E1 -1069.046,E2 -1069.046} C_VEL
LIN {X 0,Y 746.441,Z 495.258,A -85,B 0,C 180,E1 -1069.593,E2 -1069.593} C_VEL
LIN {X 0,Y 746.381,Z 506.439,A -85,B 0,C 180,E1 -1070.275,E2 -1070.275} C_VEL
LIN {X 0,Y 746.337,Z 517.456,A -85,B 0,C 180,E1 -1071.091,E2 -1071.091} C_VEL
LIN {X 0,Y 746.334,Z 527.861,A -85,B 0,C 180,E1 -1072.043,E2 -1072.043} C_VEL
LIN {X 0,Y 746.3,Z 536.261,A -85,B 0,C 180,E1 -1072.992,E2 -1072.992} C_VEL
LIN {X 0,Y 746.287,Z 542.139,A -85,B 0,C 180,E1 -1073.803,E2 -1073.803} C_VEL
LIN {X 0,Y 746.259,Z 546.983,A -85,B 0,C 180,E1 -1074.614,E2 -1074.614} C_VEL
LIN {X 0,Y 746.256,Z 550.924,A -85,B 0,C 180,E1 -1075.424,E2 -1075.424} C_VEL
LIN {X 0,Y 746.284,Z 553.951,A -85,B 0,C 180,E1 -1076.233,E2 -1076.233} C_VEL
LIN {X 0,Y 746.245,Z 556.768,A -85,B 0,C 180,E1 -1077.31,E2 -1077.31} C_VEL
LIN {X 0,Y 746.234,Z 558.232,A -85,B 0,C 180,E1 -1078.386,E2 -1078.386} C_VEL
LIN {X 0,Y 746.242,Z 558.378,A -85,B 0,C 180,E1 -1079.462,E2 -1079.462} C_VEL
LIN {X 0,Y 746.243,Z 557.213,A -85,B 0,C 180,E1 -1080.538,E2 -1080.538} C_VEL
LIN {X 0,Y 746.242,Z 554.723,A -85,B 0,C 180,E1 -1081.613,E2 -1081.613} C_VEL
LIN {X 0,Y 746.251,Z 550.822,A -85,B 0,C 180,E1 -1082.69,E2 -1082.69} C_VEL
LIN {X 0,Y 746.288,Z 545.364,A -85,B 0,C 180,E1 -1083.767,E2 -1083.767} C_VEL
LIN {X 0,Y 746.278,Z 539.199,A -85,B 0,C 180,E1 -1084.711,E2 -1084.711} C_VEL
LIN {X 0,Y 746.3,Z 531.854,A -85,B 0,C 180,E1 -1085.618,E2 -1085.618} C_VEL
LIN {X 0,Y 746.329,Z 523.513,A -85,B 0,C 180,E1 -1086.466,E2 -1086.466} C_VEL
LIN {X 0,Y 746.377,Z 513.893,A -85,B 0,C 180,E1 -1087.278,E2 -1087.278} C_VEL
LIN {X 0,Y 746.402,Z 503.232,A -85,B 0,C 180,E1 -1088.024,E2 -1088.024} C_VEL
LIN {X 0,Y 746.45,Z 491.449,A -85,B 0,C 180,E1 -1088.703,E2 -1088.703} C_VEL
LIN {X 0,Y 746.51,Z 478.242,A -85,B 0,C 180,E1 -1089.314,E2 -1089.314} C_VEL
LIN {X 0,Y 746.557,Z 464.882,A -85,B 0,C 180,E1 -1089.798,E2 -1089.798} C_VEL
LIN {X 0,Y 746.586,Z 451.609,A -85,B 0,C 180,E1 -1090.166,E2 -1090.166} C_VEL
LIN {X 0,Y 746.628,Z 437.834,A -85,B 0,C 180,E1 -1090.438,E2 -1090.438} C_VEL
LIN {X 0,Y 746.651,Z 420.382,A -85,B 0,C 180,E1 -1090.643,E2 -1090.643} C_VEL
LIN {X 0,Y 746.624,Z 306.241,A -85,B 0,C 180,E1 -1091.744,E2 -1091.744} C_VEL
LIN {X 0,Y 746.369,Z 305.068,A -85,B 0,C 180,E1 -1091.761,E2 -1091.761} C_VEL
LIN {X 0,Y 746.344,Z 305.075,A -85,B 0,C 180,E1 -1094.123,E2 -1094.123} C_VEL
LIN {X 0,Y 746.375,Z 305.077,A -85,B 0,C 180,E1 -1096.352,E2 -1096.352} C_VEL
LIN {X 0,Y 746.392,Z 305.068,A -85,B 0,C 180,E1 -1098.607,E2 -1098.607} C_VEL
LIN {X 0,Y 746.373,Z 305.065,A -85,B 0,C 180,E1 -1100.892,E2 -1100.892} C_VEL
LIN {X 0,Y 746.352,Z 305.068,A -85,B 0,C 180,E1 -1103.214,E2 -1103.214} C_VEL
LIN {X 0,Y 746.389,Z 305.071,A -85,B 0,C 180,E1 -1105.722,E2 -1105.722} C_VEL
LIN {X 0,Y 746.386,Z 305.07,A -85,B 0,C 180,E1 -1108.098,E2 -1108.098} C_VEL
LIN {X 0,Y 746.356,Z 305.068,A -85,B 0,C 180,E1 -1110.45,E2 -1110.45} C_VEL
LIN {X 0,Y 746.375,Z 305.066,A -85,B 0,C 180,E1 -1112.977,E2 -1112.977} C_VEL
LIN {X 0,Y 746.372,Z 305.075,A -85,B 0,C 180,E1 -1115.581,E2 -1115.581} C_VEL
LIN {X 0,Y 746.354,Z 305.069,A -85,B 0,C 180,E1 -1117.97,E2 -1117.97} C_VEL
LIN {X 0,Y 746.369,Z 305.065,A -85,B 0,C 180,E1 -1120.521,E2 -1120.521} C_VEL
LIN {X 0,Y 746.371,Z 305.076,A -85,B 0,C 180,E1 -1123.242,E2 -1123.242} C_VEL
LIN {X 0,Y 746.335,Z 305.073,A -85,B 0,C 180,E1 -1125.502,E2 -1125.502} C_VEL
LIN {X 0,Y 746.324,Z 305.071,A -85,B 0,C 180,E1 -1127.854,E2 -1127.854} C_VEL
LIN {X 0,Y 746.304,Z 305.074,A -85,B 0,C 180,E1 -1129.639,E2 -1129.639} C_VEL
LIN {X 0,Y 746.339,Z 305.069,A -85,B 0,C 180,E1 -1132.031,E2 -1132.031} C_VEL
LIN {X 0,Y 746.314,Z 305.078,A -85,B 0,C 180,E1 -1134.416,E2 -1134.416} C_VEL
LIN {X 0,Y 746.326,Z 305.082,A -85,B 0,C 180,E1 -1136.646,E2 -1136.646} C_VEL
LIN {X 0,Y 746.321,Z 305.076,A -85,B 0,C 180,E1 -1138.923,E2 -1138.923} C_VEL
LIN {X 0,Y 746.363,Z 305.072,A -85,B 0,C 180,E1 -1140.79,E2 -1140.79} C_VEL
LIN {X 0,Y 746.329,Z 305.071,A -85,B 0,C 180,E1 -1143.225,E2 -1143.225} C_VEL
LIN {X 0,Y 746.33,Z 305.216,A -85,B 0,C 180,E1 -1145.052,E2 -1145.052} C_VEL
LIN {X 0,Y 747.035,Z 309.226,A -85,B 0,C 180,E1 -1145.437,E2 -1145.437} C_VEL
LIN {X 0,Y 746.956,Z 335.931,A -85,B 0,C 180,E1 -1147.825,E2 -1147.825} C_VEL
LIN {X 0,Y 746.768,Z 366.991,A -85,B 0,C 180,E1 -1150.55,E2 -1150.55} C_VEL
LIN {X 0,Y 746.603,Z 394.782,A -85,B 0,C 180,E1 -1152.951,E2 -1152.951} C_VEL
LIN {X 0,Y 746.485,Z 418.989,A -85,B 0,C 180,E1 -1155.019,E2 -1155.019} C_VEL
LIN {X 0,Y 746.446,Z 443.548,A -85,B 0,C 180,E1 -1157.099,E2 -1157.099} C_VEL
LIN {X 0,Y 746.438,Z 444.567,A -85,B 0,C 180,E1 -1157.185,E2 -1157.185} C_VEL
LIN {X 0,Y 746.729,Z 452.852,A -85,B 0,C 180,E1 -1157.27,E2 -1157.27} C_VEL
LIN {X 0,Y 746.606,Z 583.002,A -85,B 0,C 180,E1 -1158.535,E2 -1158.535} C_VEL
LIN {X 0,Y 746.602,Z 597.782,A -85,B 0,C 180,E1 -1158.791,E2 -1158.791} C_VEL
LIN {X 0,Y 746.576,Z 611.791,A -85,B 0,C 180,E1 -1159.15,E2 -1159.15} C_VEL
LIN {X 0,Y 746.494,Z 624.786,A -85,B 0,C 180,E1 -1159.594,E2 -1159.594} C_VEL
LIN {X 0,Y 746.456,Z 637.724,A -85,B 0,C 180,E1 -1160.156,E2 -1160.156} C_VEL
LIN {X 0,Y 746.421,Z 650,A -85,B 0,C 180,E1 -1160.82,E2 -1160.82} C_VEL
LIN {X 0,Y 746.367,Z 660.34,A -85,B 0,C 180,E1 -1161.5,E2 -1161.5} C_VEL
LIN {X 0,Y 746.354,Z 670.636,A -85,B 0,C 180,E1 -1162.314,E2 -1162.314} C_VEL
LIN {X 0,Y 746.331,Z 679.136,A -85,B 0,C 180,E1 -1163.127,E2 -1163.127} C_VEL
LIN {X 0,Y 746.306,Z 687.263,A -85,B 0,C 180,E1 -1164.074,E2 -1164.074} C_VEL
LIN {X 0,Y 746.305,Z 692.979,A -85,B 0,C 180,E1 -1164.884,E2 -1164.884} C_VEL
LIN {X 0,Y 746.243,Z 697.643,A -85,B 0,C 180,E1 -1165.693,E2 -1165.693} C_VEL
LIN {X 0,Y 746.255,Z 702.484,A -85,B 0,C 180,E1 -1166.771,E2 -1166.771} C_VEL
LIN {X 0,Y 746.226,Z 705.851,A -85,B 0,C 180,E1 -1167.848,E2 -1167.848} C_VEL
LIN {X 0,Y 746.245,Z 707.836,A -85,B 0,C 180,E1 -1168.924,E2 -1168.924} C_VEL
LIN {X 0,Y 746.24,Z 708.5,A -85,B 0,C 180,E1 -1170,E2 -1170} C_VEL
LIN {X 0,Y 746.245,Z 707.836,A -85,B 0,C 180,E1 -1171.076,E2 -1171.076} C_VEL
LIN {X 0,Y 746.226,Z 705.85,A -85,B 0,C 180,E1 -1172.152,E2 -1172.152} C_VEL
LIN {X 0,Y 746.255,Z 702.484,A -85,B 0,C 180,E1 -1173.228,E2 -1173.228} C_VEL
LIN {X 0,Y 746.242,Z 697.645,A -85,B 0,C 180,E1 -1174.306,E2 -1174.306} C_VEL
LIN {X 0,Y 746.305,Z 692.98,A -85,B 0,C 180,E1 -1175.115,E2 -1175.115} C_VEL
LIN {X 0,Y 746.305,Z 686.207,A -85,B 0,C 180,E1 -1176.061,E2 -1176.061} C_VEL
LIN {X 0,Y 746.306,Z 677.795,A -85,B 0,C 180,E1 -1177.008,E2 -1177.008} C_VEL
LIN {X 0,Y 746.351,Z 669.024,A -85,B 0,C 180,E1 -1177.821,E2 -1177.821} C_VEL
LIN {X 0,Y 746.361,Z 658.41,A -85,B 0,C 180,E1 -1178.636,E2 -1178.636} C_VEL
LIN {X 0,Y 746.444,Z 646.522,A -85,B 0,C 180,E1 -1179.383,E2 -1179.383} C_VEL
LIN {X 0,Y 746.489,Z 635.114,A -85,B 0,C 180,E1 -1179.969,E2 -1179.969} C_VEL
LIN {X 0,Y 746.509,Z 623.037,A -85,B 0,C 180,E1 -1180.474,E2 -1180.474} C_VEL
LIN {X 0,Y 746.589,Z 609.531,A -85,B 0,C 180,E1 -1180.918,E2 -1180.918} C_VEL
LIN {X 0,Y 746.601,Z 595.33,A -85,B 0,C 180,E1 -1181.26,E2 -1181.26} C_VEL
LIN {X 0,Y 746.632,Z 581.552,A -85,B 0,C 180,E1 -1181.482,E2 -1181.482} C_VEL
LIN {X 0,Y 746.592,Z 445.562,A -85,B 0,C 180,E1 -1182.802,E2 -1182.802} C_VEL
LIN {X 0,Y 746.446,Z 444.495,A -85,B 0,C 180,E1 -1182.821,E2 -1182.821} C_VEL
LIN {X 0,Y 746.484,Z 420.197,A -85,B 0,C 180,E1 -1184.878,E2 -1184.878} C_VEL
LIN {X 0,Y 746.596,Z 396.418,A -85,B 0,C 180,E1 -1186.908,E2 -1186.908} C_VEL
LIN {X 0,Y 746.746,Z 368.628,A -85,B 0,C 180,E1 -1189.308,E2 -1189.308} C_VEL
LIN {X 0,Y 746.923,Z 339.412,A -85,B 0,C 180,E1 -1191.868,E2 -1191.868} C_VEL
LIN {X 0,Y 747.042,Z 310.394,A -85,B 0,C 180,E1 -1194.457,E2 -1194.457} C_VEL
LIN {X 0,Y 746.568,Z 306.251,A -85,B 0,C 180,E1 -1194.848,E2 -1194.848} C_VEL
LIN {X 0,Y 746.31,Z 305.079,A -85,B 0,C 180,E1 -1194.983,E2 -1194.983} C_VEL
LIN {X 0,Y 746.34,Z 305.076,A -85,B 0,C 180,E1 -1197.379,E2 -1197.379} C_VEL
LIN {X 0,Y 746.348,Z 305.075,A -85,B 0,C 180,E1 -1199.828,E2 -1199.828} C_VEL
LIN {X 0,Y 746.3,Z 305.074,A -85,B 0,C 180,E1 -1202.36,E2 -1202.36} C_VEL
LIN {X 0,Y 746.319,Z 305.074,A -85,B 0,C 180,E1 -1204.925,E2 -1204.925} C_VEL
LIN {X 0,Y 746.322,Z 305.078,A -85,B 0,C 180,E1 -1207.593,E2 -1207.593} C_VEL
LIN {X 0,Y 746.326,Z 305.075,A -85,B 0,C 180,E1 -1209.683,E2 -1209.683} C_VEL
LIN {X 0,Y 746.34,Z 305.071,A -85,B 0,C 180,E1 -1211.785,E2 -1211.785} C_VEL
LIN {X 0,Y 746.311,Z 305.072,A -85,B 0,C 180,E1 -1213.989,E2 -1213.989} C_VEL
LIN {X 0,Y 746.328,Z 305.07,A -85,B 0,C 180,E1 -1216.275,E2 -1216.275} C_VEL
LIN {X 0,Y 746.364,Z 305.077,A -85,B 0,C 180,E1 -1218.934,E2 -1218.934} C_VEL
LIN {X 0,Y 746.361,Z 305.073,A -85,B 0,C 180,E1 -1221.164,E2 -1221.164} C_VEL
LIN {X 0,Y 746.338,Z 305.069,A -85,B 0,C 180,E1 -1223.815,E2 -1223.815} C_VEL
LIN {X 0,Y 746.347,Z 305.068,A -85,B 0,C 180,E1 -1225.73,E2 -1225.73} C_VEL
LIN {X 0,Y 746.345,Z 305.068,A -85,B 0,C 180,E1 -1227.66,E2 -1227.66} C_VEL
LIN {X 0,Y 746.35,Z 305.072,A -85,B 0,C 180,E1 -1230.172,E2 -1230.172} C_VEL
LIN {X 0,Y 746.341,Z 305.081,A -85,B 0,C 180,E1 -1232.622,E2 -1232.622} C_VEL
LIN {X 0,Y 746.338,Z 305.076,A -85,B 0,C 180,E1 -1235.018,E2 -1235.018} C_VEL
LIN {X 0,Y 746.329,Z 305.078,A -85,B 0,C 180,E1 -1235.303,E2 -1235.303} C_VEL
LIN {X 0,Y 747.009,Z 308.412,A -85,B 0,C 180,E1 -1235.634,E2 -1235.634} C_VEL
LIN {X 0,Y 746.937,Z 334.093,A -85,B 0,C 180,E1 -1237.969,E2 -1237.969} C_VEL
LIN {X 0,Y 746.756,Z 362.984,A -85,B 0,C 180,E1 -1240.55,E2 -1240.55} C_VEL
LIN {X 0,Y 746.609,Z 393.392,A -85,B 0,C 180,E1 -1243.225,E2 -1243.225} C_VEL
LIN {X 0,Y 746.527,Z 420.77,A -85,B 0,C 180,E1 -1245.603,E2 -1245.603} C_VEL
LIN {X 0,Y 746.466,Z 439.639,A -85,B 0,C 180,E1 -1247.227,E2 -1247.227} C_VEL
LIN {X 0,Y 746.751,Z 449.114,A -85,B 0,C 180,E1 -1247.328,E2 -1247.328} C_VEL
LIN {X 0,Y 746.605,Z 578.372,A -85,B 0,C 180,E1 -1248.586,E2 -1248.586} C_VEL
LIN {X 0,Y 746.611,Z 592.28,A -85,B 0,C 180,E1 -1248.826,E2 -1248.826} C_VEL
LIN {X 0,Y 746.562,Z 606.464,A -85,B 0,C 180,E1 -1249.185,E2 -1249.185} C_VEL
LIN {X 0,Y 746.461,Z 620.385,A -85,B 0,C 180,E1 -1249.662,E2 -1249.662} C_VEL
LIN {X 0,Y 746.449,Z 632.97,A -85,B 0,C 180,E1 -1250.215,E2 -1250.215} C_VEL
LIN {X 0,Y 746.421,Z 644.233,A -85,B 0,C 180,E1 -1250.821,E2 -1250.821} C_VEL
LIN {X 0,Y 746.376,Z 654.709,A -85,B 0,C 180,E1 -1251.5,E2 -1251.5} C_VEL
LIN {X 0,Y 746.355,Z 665.113,A -85,B 0,C 180,E1 -1252.315,E2 -1252.315} C_VEL
LIN {X 0,Y 746.337,Z 673.685,A -85,B 0,C 180,E1 -1253.128,E2 -1253.128} C_VEL
LIN {X 0,Y 746.306,Z 681.925,A -85,B 0,C 180,E1 -1254.074,E2 -1254.074} C_VEL
LIN {X 0,Y 746.285,Z 689.359,A -85,B 0,C 180,E1 -1255.154,E2 -1255.154} C_VEL
LIN {X 0,Y 746.29,Z 695.042,A -85,B 0,C 180,E1 -1256.233,E2 -1256.233} C_VEL
LIN {X 0,Y 746.248,Z 699.196,A -85,B 0,C 180,E1 -1257.31,E2 -1257.31} C_VEL
LIN {X 0,Y 746.24,Z 701.923,A -85,B 0,C 180,E1 -1258.387,E2 -1258.387} C_VEL
LIN {X 0,Y 746.241,Z 703.299,A -85,B 0,C 180,E1 -1259.462,E2 -1259.462} C_VEL
LIN {X 0,Y 746.239,Z 703.357,A -85,B 0,C 180,E1 -1260.538,E2 -1260.538} C_VEL
LIN {X 0,Y 746.234,Z 702.094,A -85,B 0,C 180,E1 -1261.614,E2 -1261.614} C_VEL
LIN {X 0,Y 746.247,Z 699.49,A -85,B 0,C 180,E1 -1262.69,E2 -1262.69} C_VEL
LIN {X 0,Y 746.29,Z 695.452,A -85,B 0,C 180,E1 -1263.767,E2 -1263.767} C_VEL
LIN {X 0,Y 746.284,Z 689.894,A -85,B 0,C 180,E1 -1264.846,E2 -1264.846} C_VEL
LIN {X 0,Y 746.27,Z 682.605,A -85,B 0,C 180,E1 -1265.926,E2 -1265.926} C_VEL
LIN {X 0,Y 746.332,Z 674.542,A -85,B 0,C 180,E1 -1266.873,E2 -1266.873} C_VEL
LIN {X 0,Y 746.354,Z 666.117,A -85,B 0,C 180,E1 -1267.686,E2 -1267.686} C_VEL
LIN {X 0,Y 746.366,Z 655.984,A -85,B 0,C 180,E1 -1268.5,E2 -1268.5} C_VEL
LIN {X 0,Y 746.424,Z 644.601,A -85,B 0,C 180,E1 -1269.248,E2 -1269.248} C_VEL
LIN {X 0,Y 746.448,Z 632.401,A -85,B 0,C 180,E1 -1269.903,E2 -1269.903} C_VEL
LIN {X 0,Y 746.492,Z 620.932,A -85,B 0,C 180,E1 -1270.406,E2 -1270.406} C_VEL
LIN {X 0,Y 746.512,Z 615.597,A -85,B 0,C 180,E1 -1270.607,E2 -1270.607} C_VEL
LIN {X 0,Y 745.873,Z 610.257,A -85,B 0,C 180,E1 -1270.799,E2 -1270.799} C_VEL
LIN {X 0,Y 743.016,Z 601.557,A -85,B 0,C 180,E1 -1271.095,E2 -1271.095} C_VEL
LIN {X 0,Y 740.268,Z 592.661,A -85,B 0,C 180,E1 -1271.353,E2 -1271.353} C_VEL
LIN {X 0,Y 739.641,Z 587.024,A -85,B 0,C 180,E1 -1271.475,E2 -1271.475} C_VEL
LIN {X 0,Y 739.675,Z 571.389,A -85,B 0,C 180,E1 -1271.696,E2 -1271.696} C_VEL
LIN {X 0,Y 739.678,Z 441.182,A -85,B 0,C 180,E1 -1272.963,E2 -1272.963} C_VEL
LIN {X 0,Y 739.475,Z 439.682,A -85,B 0,C 180,E1 -1272.982,E2 -1272.982} C_VEL
LIN {X 0,Y 739.621,Z 410.562,A -85,B 0,C 180,E1 -1275.518,E2 -1275.518} C_VEL
LIN {X 0,Y 739.731,Z 383.261,A -85,B 0,C 180,E1 -1277.923,E2 -1277.923} C_VEL
LIN {X 0,Y 739.938,Z 354.353,A -85,B 0,C 180,E1 -1280.503,E2 -1280.503} C_VEL
LIN {X 0,Y 740.083,Z 325.888,A -85,B 0,C 180,E1 -1283.087,E2 -1283.087} C_VEL
LIN {X 0,Y 740.193,Z 310.784,A -85,B 0,C 180,E1 -1284.457,E2 -1284.457} C_VEL
LIN {X 0,Y 739.303,Z 305.953,A -85,B 0,C 180,E1 -1284.936,E2 -1284.936} C_VEL
LIN {X 0,Y 739.331,Z 305.947,A -85,B 0,C 180,E1 -1287.056,E2 -1287.056} C_VEL
LIN {X 0,Y 739.335,Z 305.952,A -85,B 0,C 180,E1 -1289.515,E2 -1289.515} C_VEL
LIN {X 0,Y 739.311,Z 305.945,A -85,B 0,C 180,E1 -1292.044,E2 -1292.044} C_VEL
LIN {X 0,Y 739.342,Z 305.941,A -85,B 0,C 180,E1 -1294.49,E2 -1294.49} C_VEL
LIN {X 0,Y 739.306,Z 305.947,A -85,B 0,C 180,E1 -1296.647,E2 -1296.647} C_VEL
LIN {X 0,Y 739.35,Z 305.95,A -85,B 0,C 180,E1 -1299.027,E2 -1299.027} C_VEL
LIN {X 0,Y 739.355,Z 305.941,A -85,B 0,C 180,E1 -1301.546,E2 -1301.546} C_VEL
LIN {X 0,Y 739.329,Z 305.942,A -85,B 0,C 180,E1 -1303.943,E2 -1303.943} C_VEL
LIN {X 0,Y 739.315,Z 305.946,A -85,B 0,C 180,E1 -1306.241,E2 -1306.241} C_VEL
LIN {X 0,Y 739.359,Z 305.944,A -85,B 0,C 180,E1 -1308.459,E2 -1308.459} C_VEL
LIN {X 0,Y 739.349,Z 305.941,A -85,B 0,C 180,E1 -1311.298,E2 -1311.298} C_VEL
LIN {X 0,Y 739.31,Z 305.944,A -85,B 0,C 180,E1 -1313.641,E2 -1313.641} C_VEL
LIN {X 0,Y 739.331,Z 305.945,A -85,B 0,C 180,E1 -1316.016,E2 -1316.016} C_VEL
LIN {X 0,Y 739.314,Z 305.952,A -85,B 0,C 180,E1 -1318.595,E2 -1318.595} C_VEL
LIN {X 0,Y 739.326,Z 305.943,A -85,B 0,C 180,E1 -1321.107,E2 -1321.107} C_VEL
LIN {X 0,Y 739.309,Z 305.946,A -85,B 0,C 180,E1 -1323.558,E2 -1323.558} C_VEL
LIN {X 0,Y 739.308,Z 305.953,A -85,B 0,C 180,E1 -1325.959,E2 -1325.959} C_VEL
LIN {X 0,Y 739.333,Z 305.948,A -85,B 0,C 180,E1 -1328.316,E2 -1328.316} C_VEL
LIN {X 0,Y 739.326,Z 305.944,A -85,B 0,C 180,E1 -1330.635,E2 -1330.635} C_VEL
LIN {X 0,Y 739.347,Z 305.94,A -85,B 0,C 180,E1 -1333.11,E2 -1333.11} C_VEL
LIN {X 0,Y 739.303,Z 305.957,A -85,B 0,C 180,E1 -1335.739,E2 -1335.739} C_VEL
LIN {X 0,Y 739.328,Z 305.949,A -85,B 0,C 180,E1 -1337.97,E2 -1337.97} C_VEL
LIN {X 0,Y 739.336,Z 305.944,A -85,B 0,C 180,E1 -1340.181,E2 -1340.181} C_VEL
LIN {X 0,Y 739.322,Z 305.947,A -85,B 0,C 180,E1 -1342.215,E2 -1342.215} C_VEL
LIN {X 0,Y 739.768,Z 308.194,A -85,B 0,C 180,E1 -1342.246,E2 -1342.246} C_VEL
LIN {X 0,Y 739.704,Z 432.977,A -85,B 0,C 180,E1 -1343.475,E2 -1343.475} C_VEL
LIN {X 0,Y 739.675,Z 445.232,A -85,B 0,C 180,E1 -1343.68,E2 -1343.68} C_VEL
LIN {X 0,Y 739.622,Z 457.033,A -85,B 0,C 180,E1 -1343.959,E2 -1343.959} C_VEL
LIN {X 0,Y 739.554,Z 468.431,A -85,B 0,C 180,E1 -1344.309,E2 -1344.309} C_VEL
LIN {X 0,Y 739.487,Z 480.339,A -85,B 0,C 180,E1 -1344.769,E2 -1344.769} C_VEL
LIN {X 0,Y 739.448,Z 491.764,A -85,B 0,C 180,E1 -1345.314,E2 -1345.314} C_VEL
LIN {X 0,Y 739.364,Z 503.474,A -85,B 0,C 180,E1 -1345.994,E2 -1345.994} C_VEL
LIN {X 0,Y 739.316,Z 515.769,A -85,B 0,C 180,E1 -1346.877,E2 -1346.877} C_VEL
LIN {X 0,Y 739.267,Z 524.997,A -85,B 0,C 180,E1 -1347.692,E2 -1347.692} C_VEL
LIN {X 0,Y 739.229,Z 532.719,A -85,B 0,C 180,E1 -1348.507,E2 -1348.507} C_VEL
LIN {X 0,Y 739.224,Z 538.183,A -85,B 0,C 180,E1 -1349.186,E2 -1349.186} C_VEL
LIN {X 0,Y 739.16,Z 543.722,A -85,B 0,C 180,E1 -1350,E2 -1350} C_VEL
LIN {X 0,Y 739.182,Z 548.264,A -85,B 0,C 180,E1 -1350.815,E2 -1350.815} C_VEL
LIN {X 0,Y 739.143,Z 551.892,A -85,B 0,C 180,E1 -1351.629,E2 -1351.629} C_VEL
LIN {X 0,Y 739.163,Z 555.45,A -85,B 0,C 180,E1 -1352.716,E2 -1352.716} C_VEL
LIN {X 0,Y 739.191,Z 557.621,A -85,B 0,C 180,E1 -1353.803,E2 -1353.803} C_VEL
LIN {X 0,Y 739.182,Z 558.459,A -85,B 0,C 180,E1 -1354.892,E2 -1354.892} C_VEL
LIN {X 0,Y 739.177,Z 557.969,A -85,B 0,C 180,E1 -1355.983,E2 -1355.983} C_VEL
LIN {X 0,Y 739.158,Z 557.273,A -85,B 0,C 180,E1 -1356.53,E2 -1356.53} C_VEL
LIN {X 0,Y 739.158,Z 554.762,A -85,B 0,C 180,E1 -1357.624,E2 -1357.624} C_VEL
LIN {X 0,Y 739.192,Z 550.798,A -85,B 0,C 180,E1 -1358.721,E2 -1358.721} C_VEL
LIN {X 0,Y 739.186,Z 547.009,A -85,B 0,C 180,E1 -1359.517,E2 -1359.517} C_VEL
LIN {X 0,Y 739.203,Z 541.906,A -85,B 0,C 180,E1 -1360.372,E2 -1360.372} C_VEL
LIN {X 0,Y 739.209,Z 534.764,A -85,B 0,C 180,E1 -1361.339,E2 -1361.339} C_VEL
LIN {X 0,Y 739.223,Z 527.264,A -85,B 0,C 180,E1 -1362.171,E2 -1362.171} C_VEL
LIN {X 0,Y 739.303,Z 519.883,A -85,B 0,C 180,E1 -1362.864,E2 -1362.864} C_VEL
LIN {X 0,Y 739.31,Z 511.191,A -85,B 0,C 180,E1 -1363.562,E2 -1363.562} C_VEL
LIN {X 0,Y 739.364,Z 500.823,A -85,B 0,C 180,E1 -1364.26,E2 -1364.26} C_VEL
LIN {X 0,Y 739.448,Z 489.755,A -85,B 0,C 180,E1 -1364.879,E2 -1364.879} C_VEL
LIN {X 0,Y 739.485,Z 478.944,A -85,B 0,C 180,E1 -1365.38,E2 -1365.38} C_VEL
LIN {X 0,Y 739.565,Z 466.823,A -85,B 0,C 180,E1 -1365.836,E2 -1365.836} C_VEL
LIN {X 0,Y 739.632,Z 454.926,A -85,B 0,C 180,E1 -1366.187,E2 -1366.187} C_VEL
LIN {X 0,Y 739.67,Z 442.234,A -85,B 0,C 180,E1 -1366.469,E2 -1366.469} C_VEL
LIN {X 0,Y 739.702,Z 427.527,A -85,B 0,C 180,E1 -1366.682,E2 -1366.682} C_VEL
LIN {X 0,Y 739.595,Z 307.367,A -85,B 0,C 180,E1 -1367.855,E2 -1367.855} C_VEL
LIN {X 0,Y 739.298,Z 305.949,A -85,B 0,C 180,E1 -1367.881,E2 -1367.881} C_VEL
LIN {X 0,Y 739.307,Z 305.953,A -85,B 0,C 180,E1 -1370.287,E2 -1370.287} C_VEL
LIN {X 0,Y 739.298,Z 305.955,A -85,B 0,C 180,E1 -1372.271,E2 -1372.271} C_VEL
LIN {X 0,Y 739.31,Z 305.953,A -85,B 0,C 180,E1 -1374.637,E2 -1374.637} C_VEL
LIN {X 0,Y 739.315,Z 305.945,A -85,B 0,C 180,E1 -1377.053,E2 -1377.053} C_VEL
LIN {X 0,Y 739.306,Z 305.945,A -85,B 0,C 180,E1 -1379.516,E2 -1379.516} C_VEL
LIN {X 0,Y 739.289,Z 305.954,A -85,B 0,C 180,E1 -1382.045,E2 -1382.045} C_VEL
LIN {X 0,Y 739.288,Z 305.952,A -85,B 0,C 180,E1 -1384.644,E2 -1384.644} C_VEL
LIN {X 0,Y 739.295,Z 305.95,A -85,B 0,C 180,E1 -1386.648,E2 -1386.648} C_VEL
LIN {X 0,Y 739.314,Z 305.944,A -85,B 0,C 180,E1 -1389.023,E2 -1389.023} C_VEL
LIN {X 0,Y 739.33,Z 305.943,A -85,B 0,C 180,E1 -1391.543,E2 -1391.543} C_VEL
LIN {X 0,Y 739.307,Z 305.954,A -85,B 0,C 180,E1 -1393.941,E2 -1393.941} C_VEL
LIN {X 0,Y 739.308,Z 305.953,A -85,B 0,C 180,E1 -1396.241,E2 -1396.241} C_VEL
LIN {X 0,Y 739.33,Z 305.945,A -85,B 0,C 180,E1 -1398.457,E2 -1398.457} C_VEL
LIN {X 0,Y 739.285,Z 305.946,A -85,B 0,C 180,E1 -1400.98,E2 -1400.98} C_VEL
LIN {X 0,Y 739.277,Z 305.948,A -85,B 0,C 180,E1 -1403.351,E2 -1403.351} C_VEL
LIN {X 0,Y 739.309,Z 305.954,A -85,B 0,C 180,E1 -1406.014,E2 -1406.014} C_VEL
LIN {X 0,Y 739.296,Z 305.945,A -85,B 0,C 180,E1 -1408.594,E2 -1408.594} C_VEL
LIN {X 0,Y 739.31,Z 305.944,A -85,B 0,C 180,E1 -1410.65,E2 -1410.65} C_VEL
LIN {X 0,Y 739.297,Z 305.945,A -85,B 0,C 180,E1 -1412.949,E2 -1412.949} C_VEL
LIN {X 0,Y 739.317,Z 305.949,A -85,B 0,C 180,E1 -1415.44,E2 -1415.44} C_VEL
LIN {X 0,Y 739.316,Z 305.944,A -85,B 0,C 180,E1 -1418.315,E2 -1418.315} C_VEL
LIN {X 0,Y 739.29,Z 305.947,A -85,B 0,C 180,E1 -1420.633,E2 -1420.633} C_VEL
LIN {X 0,Y 739.302,Z 305.949,A -85,B 0,C 180,E1 -1423.121,E2 -1423.121} C_VEL
LIN {X 0,Y 739.29,Z 305.957,A -85,B 0,C 180,E1 -1425.739,E2 -1425.739} C_VEL
LIN {X 0,Y 739.325,Z 305.945,A -85,B 0,C 180,E1 -1426.212,E2 -1426.212} C_VEL
LIN {X 0,Y 739.731,Z 309.132,A -85,B 0,C 180,E1 -1426.254,E2 -1426.254} C_VEL
LIN {X 0,Y 739.716,Z 433.104,A -85,B 0,C 180,E1 -1427.473,E2 -1427.473} C_VEL
LIN {X 0,Y 739.65,Z 447.068,A -85,B 0,C 180,E1 -1427.715,E2 -1427.715} C_VEL
LIN {X 0,Y 739.581,Z 460.125,A -85,B 0,C 180,E1 -1428.043,E2 -1428.043} C_VEL
LIN {X 0,Y 739.533,Z 472.62,A -85,B 0,C 180,E1 -1428.458,E2 -1428.458} C_VEL
LIN {X 0,Y 739.498,Z 484.214,A -85,B 0,C 180,E1 -1428.942,E2 -1428.942} C_VEL
LIN {X 0,Y 739.412,Z 495.071,A -85,B 0,C 180,E1 -1429.493,E2 -1429.493} C_VEL
LIN {X 0,Y 739.351,Z 505.905,A -85,B 0,C 180,E1 -1430.156,E2 -1430.156} C_VEL
LIN {X 0,Y 739.326,Z 515.623,A -85,B 0,C 180,E1 -1430.869,E2 -1430.869} C_VEL
LIN {X 0,Y 739.27,Z 525.017,A -85,B 0,C 180,E1 -1431.692,E2 -1431.692} C_VEL
LIN {X 0,Y 739.221,Z 533.967,A -85,B 0,C 180,E1 -1432.651,E2 -1432.651} C_VEL
LIN {X 0,Y 739.192,Z 540.265,A -85,B 0,C 180,E1 -1433.471,E2 -1433.471} C_VEL
LIN {X 0,Y 739.168,Z 546.933,A -85,B 0,C 180,E1 -1434.562,E2 -1434.562} C_VEL
LIN {X 0,Y 739.172,Z 550.884,A -85,B 0,C 180,E1 -1435.38,E2 -1435.38} C_VEL
LIN {X 0,Y 739.191,Z 553.924,A -85,B 0,C 180,E1 -1436.197,E2 -1436.197} C_VEL
LIN {X 0,Y 739.163,Z 556.752,A -85,B 0,C 180,E1 -1437.284,E2 -1437.284} C_VEL
LIN {X 0,Y 739.134,Z 558.225,A -85,B 0,C 180,E1 -1438.371,E2 -1438.371} C_VEL
LIN {X 0,Y 739.142,Z 558.372,A -85,B 0,C 180,E1 -1439.457,E2 -1439.457} C_VEL
LIN {X 0,Y 739.143,Z 557.218,A -85,B 0,C 180,E1 -1440.543,E2 -1440.543} C_VEL
LIN {X 0,Y 739.142,Z 554.739,A -85,B 0,C 180,E1 -1441.629,E2 -1441.629} C_VEL
LIN {X 0,Y 739.172,Z 550.863,A -85,B 0,C 180,E1 -1442.716,E2 -1442.716} C_VEL
LIN {X 0,Y 739.219,Z 545.42,A -85,B 0,C 180,E1 -1443.803,E2 -1443.803} C_VEL
LIN {X 0,Y 739.203,Z 539.266,A -85,B 0,C 180,E1 -1444.756,E2 -1444.756} C_VEL
LIN {X 0,Y 739.237,Z 532.753,A -85,B 0,C 180,E1 -1445.581,E2 -1445.581} C_VEL
LIN {X 0,Y 739.271,Z 525.077,A -85,B 0,C 180,E1 -1446.392,E2 -1446.392} C_VEL
LIN {X 0,Y 739.332,Z 515.746,A -85,B 0,C 180,E1 -1447.211,E2 -1447.211} C_VEL
LIN {X 0,Y 739.369,Z 505.451,A -85,B 0,C 180,E1 -1447.964,E2 -1447.964} C_VEL
LIN {X 0,Y 739.425,Z 494.154,A -85,B 0,C 180,E1 -1448.649,E2 -1448.649} C_VEL
LIN {X 0,Y 739.507,Z 481.645,A -85,B 0,C 180,E1 -1449.266,E2 -1449.266} C_VEL
LIN {X 0,Y 739.552,Z 467.555,A -85,B 0,C 180,E1 -1449.816,E2 -1449.816} C_VEL
LIN {X 0,Y 739.627,Z 453.2,A -85,B 0,C 180,E1 -1450.233,E2 -1450.233} C_VEL
LIN {X 0,Y 739.684,Z 439.549,A -85,B 0,C 180,E1 -1450.52,E2 -1450.52} C_VEL
LIN {X 0,Y 739.714,Z 424.894,A -85,B 0,C 180,E1 -1450.71,E2 -1450.71} C_VEL
LIN {X 0,Y 739.756,Z 307.637,A -85,B 0,C 180,E1 -1451.85,E2 -1451.85} C_VEL
LIN {X 0,Y 739.35,Z 305.944,A -85,B 0,C 180,E1 -1451.874,E2 -1451.874} C_VEL
LIN {X 0,Y 739.304,Z 305.955,A -85,B 0,C 180,E1 -1454.261,E2 -1454.261} C_VEL
LIN {X 0,Y 739.346,Z 305.943,A -85,B 0,C 180,E1 -1456.89,E2 -1456.89} C_VEL
LIN {X 0,Y 739.334,Z 305.942,A -85,B 0,C 180,E1 -1459.365,E2 -1459.365} C_VEL
LIN {X 0,Y 739.32,Z 305.95,A -85,B 0,C 180,E1 -1461.802,E2 -1461.802} C_VEL
LIN {X 0,Y 739.31,Z 305.957,A -85,B 0,C 180,E1 -1464.041,E2 -1464.041} C_VEL
LIN {X 0,Y 739.305,Z 305.948,A -85,B 0,C 180,E1 -1466.442,E2 -1466.442} C_VEL
LIN {X 0,Y 739.346,Z 305.94,A -85,B 0,C 180,E1 -1468.892,E2 -1468.892} C_VEL
LIN {X 0,Y 739.314,Z 305.952,A -85,B 0,C 180,E1 -1471.495,E2 -1471.495} C_VEL
LIN {X 0,Y 739.323,Z 305.947,A -85,B 0,C 180,E1 -1473.985,E2 -1473.985} C_VEL
LIN {X 0,Y 739.302,Z 305.945,A -85,B 0,C 180,E1 -1476.358,E2 -1476.358} C_VEL
LIN {X 0,Y 739.345,Z 305.945,A -85,B 0,C 180,E1 -1479.026,E2 -1479.026} C_VEL
LIN {X 0,Y 739.328,Z 305.948,A -85,B 0,C 180,E1 -1481.543,E2 -1481.543} C_VEL
LIN {X 0,Y 739.308,Z 305.945,A -85,B 0,C 180,E1 -1483.941,E2 -1483.941} C_VEL
LIN {X 0,Y 739.297,Z 305.946,A -85,B 0,C 180,E1 -1486.24,E2 -1486.24} C_VEL
LIN {X 0,Y 739.328,Z 305.945,A -85,B 0,C 180,E1 -1488.456,E2 -1488.456} C_VEL
LIN {X 0,Y 739.326,Z 305.946,A -85,B 0,C 180,E1 -1491.296,E2 -1491.296} C_VEL
LIN {X 0,Y 739.265,Z 305.95,A -85,B 0,C 180,E1 -1493.646,E2 -1493.646} C_VEL
LIN {X 0,Y 739.292,Z 305.948,A -85,B 0,C 180,E1 -1496.013,E2 -1496.013} C_VEL
LIN {X 0,Y 739.288,Z 305.959,A -85,B 0,C 180,E1 -1498.594,E2 -1498.594} C_VEL
LIN {X 0,Y 739.298,Z 305.948,A -85,B 0,C 180,E1 -1501.105,E2 -1501.105} C_VEL
LIN {X 0,Y 739.269,Z 305.952,A -85,B 0,C 180,E1 -1503.556,E2 -1503.556} C_VEL
LIN {X 0,Y 739.279,Z 305.969,A -85,B 0,C 180,E1 -1504.932,E2 -1504.932} C_VEL
LIN {X 0,Y 740.166,Z 311.006,A -85,B 0,C 180,E1 -1505.393,E2 -1505.393} C_VEL
LIN {X 0,Y 740.086,Z 329.606,A -85,B 0,C 180,E1 -1507.039,E2 -1507.039} C_VEL
LIN {X 0,Y 739.969,Z 352.278,A -85,B 0,C 180,E1 -1509.063,E2 -1509.063} C_VEL
LIN {X 0,Y 739.773,Z 380.28,A -85,B 0,C 180,E1 -1511.525,E2 -1511.525} C_VEL
LIN {X 0,Y 739.631,Z 409.494,A -85,B 0,C 180,E1 -1514.06,E2 -1514.06} C_VEL
LIN {X 0,Y 739.471,Z 437.285,A -85,B 0,C 180,E1 -1516.441,E2 -1516.441} C_VEL
LIN {X 0,Y 739.427,Z 444.549,A -85,B 0,C 180,E1 -1517.06,E2 -1517.06} C_VEL
LIN {X 0,Y 739.834,Z 450.875,A -85,B 0,C 180,E1 -1517.131,E2 -1517.131} C_VEL
LIN {X 0,Y 739.657,Z 583.001,A -85,B 0,C 180,E1 -1518.425,E2 -1518.425} C_VEL
LIN {X 0,Y 739.663,Z 597.021,A -85,B 0,C 180,E1 -1518.668,E2 -1518.668} C_VEL
LIN {X 0,Y 739.606,Z 610.664,A -85,B 0,C 180,E1 -1519.012,E2 -1519.012} C_VEL
LIN {X 0,Y 739.523,Z 623.03,A -85,B 0,C 180,E1 -1519.425,E2 -1519.425} C_VEL
LIN {X 0,Y 739.473,Z 635.967,A -85,B 0,C 180,E1 -1519.977,E2 -1519.977} C_VEL
LIN {X 0,Y 739.419,Z 647.788,A -85,B 0,C 180,E1 -1520.601,E2 -1520.601} C_VEL
LIN {X 0,Y 739.325,Z 658.409,A -85,B 0,C 180,E1 -1521.281,E2 -1521.281} C_VEL
LIN {X 0,Y 739.288,Z 669.022,A -85,B 0,C 180,E1 -1522.104,E2 -1522.104} C_VEL
LIN {X 0,Y 739.256,Z 677.794,A -85,B 0,C 180,E1 -1522.925,E2 -1522.925} C_VEL
LIN {X 0,Y 739.239,Z 686.205,A -85,B 0,C 180,E1 -1523.881,E2 -1523.881} C_VEL
LIN {X 0,Y 739.215,Z 692.978,A -85,B 0,C 180,E1 -1524.835,E2 -1524.835} C_VEL
LIN {X 0,Y 739.15,Z 697.644,A -85,B 0,C 180,E1 -1525.652,E2 -1525.652} C_VEL
LIN {X 0,Y 739.159,Z 701.43,A -85,B 0,C 180,E1 -1526.469,E2 -1526.469} C_VEL
LIN {X 0,Y 739.166,Z 704.346,A -85,B 0,C 180,E1 -1527.284,E2 -1527.284} C_VEL
LIN {X 0,Y 739.138,Z 707.012,A -85,B 0,C 180,E1 -1528.371,E2 -1528.371} C_VEL
LIN {X 0,Y 739.14,Z 708.334,A -85,B 0,C 180,E1 -1529.457,E2 -1529.457} C_VEL
LIN {X 0,Y 739.14,Z 708.334,A -85,B 0,C 180,E1 -1530.543,E2 -1530.543} C_VEL
LIN {X 0,Y 739.138,Z 707.011,A -85,B 0,C 180,E1 -1531.629,E2 -1531.629} C_VEL
LIN {X 0,Y 739.166,Z 704.345,A -85,B 0,C 180,E1 -1532.716,E2 -1532.716} C_VEL
LIN {X 0,Y 739.22,Z 700.257,A -85,B 0,C 180,E1 -1533.803,E2 -1533.803} C_VEL
LIN {X 0,Y 739.212,Z 694.625,A -85,B 0,C 180,E1 -1534.892,E2 -1534.892} C_VEL
LIN {X 0,Y 739.188,Z 688.975,A -85,B 0,C 180,E1 -1535.751,E2 -1535.751} C_VEL
LIN {X 0,Y 739.25,Z 681.611,A -85,B 0,C 180,E1 -1536.665,E2 -1536.665} C_VEL
LIN {X 0,Y 739.293,Z 672.13,A -85,B 0,C 180,E1 -1537.622,E2 -1537.622} C_VEL
LIN {X 0,Y 739.322,Z 662.207,A -85,B 0,C 180,E1 -1538.444,E2 -1538.444} C_VEL
LIN {X 0,Y 739.377,Z 651.158,A -85,B 0,C 180,E1 -1539.199,E2 -1539.199} C_VEL
LIN {X 0,Y 739.467,Z 640.182,A -85,B 0,C 180,E1 -1539.817,E2 -1539.817} C_VEL
LIN {X 0,Y 739.506,Z 628.272,A -85,B 0,C 180,E1 -1540.368,E2 -1540.368} C_VEL
LIN {X 0,Y 739.582,Z 615.155,A -85,B 0,C 180,E1 -1540.85,E2 -1540.85} C_VEL
LIN {X 0,Y 739.646,Z 601.582,A -85,B 0,C 180,E1 -1541.229,E2 -1541.229} C_VEL
LIN {X 0,Y 739.641,Z 587.605,A -85,B 0,C 180,E1 -1541.506,E2 -1541.506} C_VEL
LIN {X 0,Y 739.712,Z 569.996,A -85,B 0,C 180,E1 -1541.712,E2 -1541.712} C_VEL
LIN {X 0,Y 739.731,Z 446.716,A -85,B 0,C 180,E1 -1542.912,E2 -1542.912} C_VEL
LIN {X 0,Y 739.434,Z 444.488,A -85,B 0,C 180,E1 -1542.945,E2 -1542.945} C_VEL
LIN {X 0,Y 739.502,Z 420.969,A -85,B 0,C 180,E1 -1544.955,E2 -1544.955} C_VEL
LIN {X 0,Y 739.689,Z 394.784,A -85,B 0,C 180,E1 -1547.213,E2 -1547.213} C_VEL
LIN {X 0,Y 739.881,Z 365.358,A -85,B 0,C 180,E1 -1549.782,E2 -1549.782} C_VEL
LIN {X 0,Y 740.104,Z 335.933,A -85,B 0,C 180,E1 -1552.391,E2 -1552.391} C_VEL
LIN {X 0,Y 740.183,Z 312.726,A -85,B 0,C 180,E1 -1554.457,E2 -1554.457} C_VEL
LIN {X 0,Y 739.885,Z 308.767,A -85,B 0,C 180,E1 -1554.809,E2 -1554.809} C_VEL
LIN {X 0,Y 739.272,Z 305.957,A -85,B 0,C 180,E1 -1555.087,E2 -1555.087} C_VEL
LIN {X 0,Y 739.293,Z 305.949,A -85,B 0,C 180,E1 -1557.051,E2 -1557.051} C_VEL
LIN {X 0,Y 739.321,Z 305.954,A -85,B 0,C 180,E1 -1559.515,E2 -1559.515} C_VEL
LIN {X 0,Y 739.262,Z 305.953,A -85,B 0,C 180,E1 -1562.046,E2 -1562.046} C_VEL
LIN {X 0,Y 739.278,Z 305.948,A -85,B 0,C 180,E1 -1564.482,E2 -1564.482} C_VEL
LIN {X 0,Y 739.307,Z 305.955,A -85,B 0,C 180,E1 -1567.265,E2 -1567.265} C_VEL
LIN {X 0,Y 739.275,Z 305.951,A -85,B 0,C 180,E1 -1569.874,E2 -1569.874} C_VEL
LIN {X 0,Y 739.27,Z 305.949,A -85,B 0,C 180,E1 -1572.277,E2 -1572.277} C_VEL
LIN {X 0,Y 739.295,Z 305.951,A -85,B 0,C 180,E1 -1574.717,E2 -1574.717} C_VEL
LIN {X 0,Y 739.282,Z 305.959,A -85,B 0,C 180,E1 -1576.986,E2 -1576.986} C_VEL
LIN {X 0,Y 739.32,Z 305.95,A -85,B 0,C 180,E1 -1579.283,E2 -1579.283} C_VEL
LIN {X 0,Y 739.322,Z 305.948,A -85,B 0,C 180,E1 -1581.296,E2 -1581.296} C_VEL
LIN {X 0,Y 739.291,Z 305.947,A -85,B 0,C 180,E1 -1583.643,E2 -1583.643} C_VEL
LIN {X 0,Y 739.307,Z 305.946,A -85,B 0,C 180,E1 -1586.014,E2 -1586.014} C_VEL
LIN {X 0,Y 739.306,Z 305.956,A -85,B 0,C 180,E1 -1588.595,E2 -1588.595} C_VEL
LIN {X 0,Y 739.329,Z 305.947,A -85,B 0,C 180,E1 -1591.107,E2 -1591.107} C_VEL
LIN {X 0,Y 739.288,Z 305.948,A -85,B 0,C 180,E1 -1593.557,E2 -1593.557} C_VEL
LIN {X 0,Y 739.301,Z 306.056,A -85,B 0,C 180,E1 -1595.223,E2 -1595.223} C_VEL
LIN {X 0,Y 740.13,Z 311.249,A -85,B 0,C 180,E1 -1595.69,E2 -1595.69} C_VEL
LIN {X 0,Y 740.089,Z 326.26,A -85,B 0,C 180,E1 -1597.038,E2 -1597.038} C_VEL
LIN {X 0,Y 739.935,Z 351.754,A -85,B 0,C 180,E1 -1599.352,E2 -1599.352} C_VEL
LIN {X 0,Y 739.739,Z 377.564,A -85,B 0,C 180,E1 -1601.66,E2 -1601.66} C_VEL
LIN {X 0,Y 739.599,Z 403.118,A -85,B 0,C 180,E1 -1603.918,E2 -1603.918} C_VEL
LIN {X 0,Y 739.513,Z 430.407,A -85,B 0,C 180,E1 -1606.303,E2 -1606.303} C_VEL
LIN {X 0,Y 739.471,Z 439.661,A -85,B 0,C 180,E1 -1607.106,E2 -1607.106} C_VEL
LIN {X 0,Y 739.84,Z 446.879,A -85,B 0,C 180,E1 -1607.185,E2 -1607.185} C_VEL
LIN {X 0,Y 739.673,Z 578.362,A -85,B 0,C 180,E1 -1608.478,E2 -1608.478} C_VEL
LIN {X 0,Y 739.635,Z 592.267,A -85,B 0,C 180,E1 -1608.719,E2 -1608.719} C_VEL
LIN {X 0,Y 739.601,Z 606.485,A -85,B 0,C 180,E1 -1609.082,E2 -1609.082} C_VEL
LIN {X 0,Y 739.481,Z 620.398,A -85,B 0,C 180,E1 -1609.563,E2 -1609.563} C_VEL
LIN {X 0,Y 739.431,Z 632.946,A -85,B 0,C 180,E1 -1610.12,E2 -1610.12} C_VEL
LIN {X 0,Y 739.398,Z 644.24,A -85,B 0,C 180,E1 -1610.733,E2 -1610.733} C_VEL
LIN {X 0,Y 739.342,Z 654.719,A -85,B 0,C 180,E1 -1611.419,E2 -1611.419} C_VEL
LIN {X 0,Y 739.285,Z 665.114,A -85,B 0,C 180,E1 -1612.241,E2 -1612.241} C_VEL
LIN {X 0,Y 739.272,Z 673.68,A -85,B 0,C 180,E1 -1613.062,E2 -1613.062} C_VEL
LIN {X 0,Y 739.236,Z 681.922,A -85,B 0,C 180,E1 -1614.017,E2 -1614.017} C_VEL
LIN {X 0,Y 739.218,Z 687.676,A -85,B 0,C 180,E1 -1614.836,E2 -1614.836} C_VEL
LIN {X 0,Y 739.202,Z 693.809,A -85,B 0,C 180,E1 -1615.925,E2 -1615.925} C_VEL
LIN {X 0,Y 739.164,Z 697.319,A -85,B 0,C 180,E1 -1616.741,E2 -1616.741} C_VEL
LIN {X 0,Y 739.13,Z 700.733,A -85,B 0,C 180,E1 -1617.828,E2 -1617.828} C_VEL
LIN {X 0,Y 739.151,Z 702.78,A -85,B 0,C 180,E1 -1618.914,E2 -1618.914} C_VEL
LIN {X 0,Y 739.139,Z 703.493,A -85,B 0,C 180,E1 -1620,E2 -1620} C_VEL
LIN {X 0,Y 739.15,Z 702.886,A -85,B 0,C 180,E1 -1621.086,E2 -1621.086} C_VEL
LIN {X 0,Y 739.128,Z 700.96,A -85,B 0,C 180,E1 -1622.173,E2 -1622.173} C_VEL
LIN {X 0,Y 739.164,Z 697.666,A -85,B 0,C 180,E1 -1623.26,E2 -1623.26} C_VEL
LIN {X 0,Y 739.151,Z 692.884,A -85,B 0,C 180,E1 -1624.348,E2 -1624.348} C_VEL
LIN {X 0,Y 739.216,Z 688.269,A -85,B 0,C 180,E1 -1625.165,E2 -1625.165} C_VEL
LIN {X 0,Y 739.242,Z 681.545,A -85,B 0,C 180,E1 -1626.119,E2 -1626.119} C_VEL
LIN {X 0,Y 739.256,Z 673.235,A -85,B 0,C 180,E1 -1627.076,E2 -1627.076} C_VEL
LIN {X 0,Y 739.287,Z 664.567,A -85,B 0,C 180,E1 -1627.897,E2 -1627.897} C_VEL
LIN {X 0,Y 739.325,Z 654.05,A -85,B 0,C 180,E1 -1628.719,E2 -1628.719} C_VEL
LIN {X 0,Y 739.425,Z 642.458,A -85,B 0,C 180,E1 -1629.462,E2 -1629.462} C_VEL
LIN {X 0,Y 739.45,Z 631.852,A -85,B 0,C 180,E1 -1630.024,E2 -1630.024} C_VEL
LIN {X 0,Y 739.531,Z 619.18,A -85,B 0,C 180,E1 -1630.574,E2 -1630.574} C_VEL
LIN {X 0,Y 739.607,Z 604.834,A -85,B 0,C 180,E1 -1631.057,E2 -1631.057} C_VEL
LIN {X 0,Y 739.649,Z 590.766,A -85,B 0,C 180,E1 -1631.402,E2 -1631.402} C_VEL
LIN {X 0,Y 739.641,Z 587.024,A -85,B 0,C 180,E1 -1631.475,E2 -1631.475} C_VEL
LIN {X 0,Y 739.043,Z 581.312,A -85,B 0,C 180,E1 -1631.582,E2 -1631.582} C_VEL
LIN {X 0,Y 733.462,Z 562.681,A -85,B 0,C 180,E1 -1631.883,E2 -1631.883} C_VEL
LIN {X 0,Y 732.772,Z 556.871,A -85,B 0,C 180,E1 -1631.949,E2 -1631.949} C_VEL
LIN {X 0,Y 732.764,Z 442.088,A -85,B 0,C 180,E1 -1633.078,E2 -1633.078} C_VEL
LIN {X 0,Y 732.464,Z 439.582,A -85,B 0,C 180,E1 -1633.117,E2 -1633.117} C_VEL
LIN {X 0,Y 732.636,Z 410.557,A -85,B 0,C 180,E1 -1635.67,E2 -1635.67} C_VEL
LIN {X 0,Y 732.803,Z 384.862,A -85,B 0,C 180,E1 -1637.955,E2 -1637.955} C_VEL
LIN {X 0,Y 733.056,Z 354.348,A -85,B 0,C 180,E1 -1640.704,E2 -1640.704} C_VEL
LIN {X 0,Y 733.223,Z 326.122,A -85,B 0,C 180,E1 -1643.273,E2 -1643.273} C_VEL
LIN {X 0,Y 733.32,Z 312.366,A -85,B 0,C 180,E1 -1644.518,E2 -1644.518} C_VEL
LIN {X 0,Y 732.285,Z 306.829,A -85,B 0,C 180,E1 -1645.06,E2 -1645.06} C_VEL
